KUKA KRL program: MyProgram_097().src

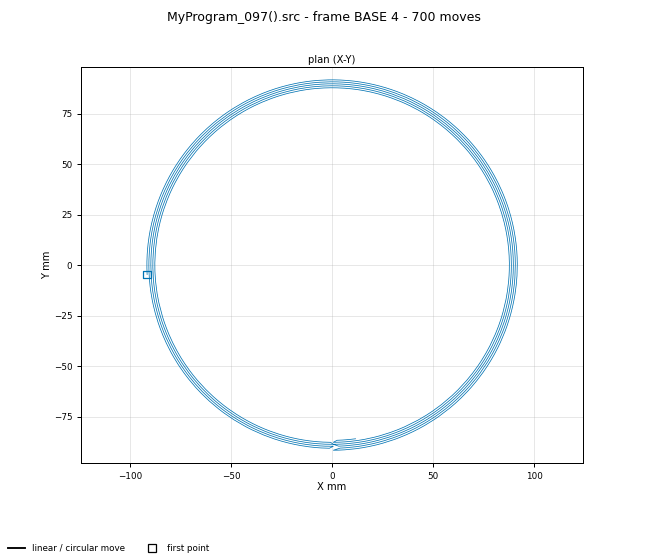
[picture p0: tool path of MyProgram_097().src in frame BASE 4, 700 of 700 moves have a stored position in this frame; points joined in program order, loops and branches not executed]
&ACCESS RVP
&REL 1
&PARAM TEMPLATE = C:\KRC\Roboter\Template\vorgabe
&PARAM EDITMASK = *
DEF MyProgram_097()
; ---- Setting reference (Base) ----
$BASE = BASE_DATA[4]

; --------------------------
; ---- Setting tool (TCP) ----
$TOOL = TOOL_DATA[3]
; --------------------------

$VEL.CP = VEL_APROX_PRINT
Startdeposition()
$VEL.CP = VEL_PRINT
LIN {X -91.5552,Y -4.6883,Z 90,A 177.5634,B 24.9231,C -2.0253,E1 24.8399,E2 -92.3942} C_DIS
LIN {X -91.6643,Y -1.3887,Z 90,A 175.5409,B 24.9225,C -2.0331,E1 24.8398,E2 -90.3782} C_DIS
LIN {X -91.6586,Y 1.702,Z 90,A 173.5845,B 24.9221,C -2.0386,E1 24.8398,E2 -88.423} C_DIS
LIN {X -91.5223,Y 5.2832,Z 90,A 171.2995,B 24.9216,C -2.0444,E1 24.8401,E2 -86.1382} C_DIS
LIN {X -91.3286,Y 7.9677,Z 90,A 169.5918,B 24.9213,C -2.049,E1 24.8405,E2 -84.4312} C_DIS
LIN {X -91.0724,Y 10.4899,Z 90,A 167.9958,B 24.9209,C -2.0538,E1 24.841,E2 -82.837} C_DIS
LIN {X -90.567,Y 14.2076,Z 90,A 165.8073,B 24.92,C -2.0659,E1 24.8419,E2 -80.6644} C_DIS
LIN {X -90.0282,Y 17.295,Z 90,A 163.689,B 24.9198,C -2.0674,E1 24.843,E2 -78.5372} C_DIS
LIN {X -89.2955,Y 20.7489,Z 90,A 161.221,B 24.9199,C -2.0667,E1 24.8445,E2 -76.0529} C_DIS
LIN {X -88.1916,Y 25.0287,Z 90,A 158.7468,B 24.9186,C -2.0839,E1 24.8463,E2 -73.6054} C_DIS
LIN {X -87.1683,Y 28.3884,Z 90,A 155.9671,B 24.9194,C -2.0734,E1 24.8486,E2 -70.7848} C_DIS
LIN {X -86.029,Y 31.6746,Z 90,A 154.4192,B 24.9174,C -2.0987,E1 24.8501,E2 -69.2883} C_DIS
LIN {X -84.932,Y 34.5072,Z 90,A 152.4774,B 24.917,C -2.1032,E1 24.8521,E2 -67.3464} C_DIS
LIN {X -83.7402,Y 37.3084,Z 90,A 150.1569,B 24.9176,C -2.0965,E1 24.8547,E2 -64.9971} C_DIS
LIN {X -81.9719,Y 41.048,Z 90,A 147.8126,B 24.9164,C -2.1113,E1 24.8575,E2 -62.6754} C_DIS
LIN {X -80.4271,Y 43.9975,Z 90,A 145.3042,B 24.9169,C -2.1046,E1 24.8609,E2 -60.138} C_DIS
LIN {X -78.8019,Y 46.8455,Z 90,A 143.8579,B 24.915,C -2.1285,E1 24.8629,E2 -58.7411} C_DIS
LIN {X -77.2171,Y 49.4139,Z 90,A 141.8308,B 24.915,C -2.1296,E1 24.8659,E2 -56.7062} C_DIS
LIN {X -75.2511,Y 52.359,Z 90,A 139.693,B 24.9143,C -2.1379,E1 24.8692,E2 -54.5777} C_DIS
LIN {X -73.255,Y 55.1171,Z 90,A 137.652,B 24.9136,C -2.1463,E1 24.8726,E2 -52.5468} C_DIS
LIN {X -71.7232,Y 57.097,Z 90,A 135.3366,B 24.9151,C -2.1278,E1 24.8767,E2 -50.1765} C_DIS
LIN {X -69.4479,Y 59.8451,Z 90,A 133.6906,B 24.9132,C -2.1511,E1 24.8796,E2 -48.5784} C_DIS
LIN {X -67.0511,Y 62.5179,Z 90,A 131.4415,B 24.9128,C -2.1565,E1 24.8838,E2 -46.3323} C_DIS
LIN {X -64.969,Y 64.6788,Z 90,A 129.4486,B 24.9127,C -2.1575,E1 24.8877,E2 -44.3333} C_DIS
LIN {X -61.8992,Y 67.6216,Z 90,A 126.93,B 24.9118,C -2.168,E1 24.8928,E2 -41.8292} C_DIS
LIN {X -59.0628,Y 70.1145,Z 90,A 124.575,B 24.9114,C -2.1734,E1 24.8978,E2 -39.478} C_DIS
LIN {X -56.7745,Y 71.9782,Z 90,A 122.6887,B 24.9112,C -2.1761,E1 24.9019,E2 -37.5911} C_DIS
LIN {X -53.5559,Y 74.405,Z 90,A 120.329,B 24.9103,C -2.1862,E1 24.9071,E2 -35.2471} C_DIS
LIN {X -51.2942,Y 75.981,Z 90,A 118.4347,B 24.9105,C -2.1844,E1 24.9115,E2 -33.3419} C_DIS
LIN {X -48.8009,Y 77.6063,Z 90,A 116.5005,B 24.9105,C -2.1856,E1 24.9161,E2 -31.4044} C_DIS
LIN {X -44.0262,Y 80.4115,Z 90,A 113.1858,B 24.9095,C -2.1962,E1 24.9241,E2 -28.1052} C_DIS
LIN {X -41.4285,Y 81.78,Z 90,A 111.0703,B 24.91,C -2.1905,E1 24.9293,E2 -25.9703} C_DIS
LIN {X -38.1771,Y 83.3487,Z 90,A 108.4553,B 24.9106,C -2.1828,E1 24.936,E2 -23.3304} C_DIS
LIN {X -34.3452,Y 84.9979,Z 90,A 106.2377,B 24.9093,C -2.1986,E1 24.9417,E2 -21.1455} C_DIS
LIN {X -31.2892,Y 86.1696,Z 90,A 104.1979,B 24.9091,C -2.2015,E1 24.947,E2 -19.1082} C_DIS
LIN {X -28.0201,Y 87.2875,Z 90,A 102.0825,B 24.9088,C -2.2055,E1 24.9526,E2 -16.9983} C_DIS
LIN {X -24.8875,Y 88.2316,Z 90,A 100.0462,B 24.9086,C -2.2079,E1 24.958,E2 -14.9646} C_DIS
LIN {X -21.729,Y 89.062,Z 90,A 97.9504,B 24.9086,C -2.2082,E1 24.9637,E2 -12.8664} C_DIS
LIN {X -18.0864,Y 89.8732,Z 90,A 95.8183,B 24.9078,C -2.2166,E1 24.9695,E2 -10.7517} C_DIS
LIN {X -15.7712,Y 90.3088,Z 90,A 94.2067,B 24.9081,C -2.2133,E1 24.9739,E2 -9.1304} C_DIS
LIN {X -12.884,Y 90.7645,Z 90,A 92.4079,B 24.9079,C -2.2154,E1 24.9789,E2 -7.3352} C_DIS
LIN {X -9.9586,Y 91.1328,Z 90,A 90.491,B 24.908,C -2.214,E1 24.9842,E2 -5.4138} C_DIS
LIN {X -6.8158,Y 91.4219,Z 90,A 87.5202,B 24.9106,C -2.1828,E1 24.9927,E2 -2.3677} C_DIS
LIN {X -1.8331,Y 91.6561,Z 90,A 85.4521,B 24.9078,C -2.2176,E1 24.9982,E2 -0.3819} C_DIS
LIN {X 0.9871,Y 91.67,Z 90,A 83.6399,B 24.9078,C -2.2163,E1 25.0033,E2 1.4333} C_DIS
LIN {X 4.2039,Y 91.5783,Z 90,A 81.6417,B 24.9078,C -2.2169,E1 25.0089,E2 3.4296} C_DIS
LIN {X 7.3964,Y 91.3755,Z 90,A 79.5848,B 24.908,C -2.2149,E1 25.0146,E2 5.4903} C_DIS
LIN {X 10.7821,Y 91.0382,Z 90,A 77.5651,B 24.9077,C -2.2181,E1 25.0202,E2 7.501} C_DIS
LIN {X 14.1056,Y 90.5827,Z 90,A 75.4649,B 24.9077,C -2.2175,E1 25.026,E2 9.6009} C_DIS
LIN {X 17.533,Y 89.9823,Z 90,A 73.3239,B 24.9077,C -2.2177,E1 25.0319,E2 11.7388} C_DIS
LIN {X 20.388,Y 89.3789,Z 90,A 71.448,B 24.908,C -2.2151,E1 25.037,E2 13.6184} C_DIS
LIN {X 23.2363,Y 88.6815,Z 90,A 69.5392,B 24.9083,C -2.2114,E1 25.0422,E2 15.5331} C_DIS
LIN {X 26.6555,Y 87.715,Z 90,A 67.2673,B 24.9085,C -2.2081,E1 25.0483,E2 17.8089} C_DIS
LIN {X 29.2709,Y 86.8758,Z 90,A 65.6725,B 24.9083,C -2.2109,E1 25.0525,E2 19.3942} C_DIS
LIN {X 32.3826,Y 85.7646,Z 90,A 63.643,B 24.9083,C -2.2102,E1 25.0578,E2 21.421} C_DIS
LIN {X 35.1234,Y 84.6806,Z 90,A 61.3887,B 24.9097,C -2.1943,E1 25.0637,E2 23.7079} C_DIS
LIN {X 39.3103,Y 82.8196,Z 90,A 58.6647,B 24.9096,C -2.1957,E1 25.0706,E2 26.4216} C_DIS
LIN {X 42.8304,Y 81.0541,Z 90,A 56.5031,B 24.909,C -2.2028,E1 25.0759,E2 28.5604} C_DIS
LIN {X 45.6049,Y 79.526,Z 90,A 54.4378,B 24.9095,C -2.1971,E1 25.081,E2 30.6331} C_DIS
LIN {X 48.5057,Y 77.7907,Z 90,A 52.3751,B 24.9095,C -2.1957,E1 25.0859,E2 32.6927} C_DIS
LIN {X 51.857,Y 75.5998,Z 90,A 50.0088,B 24.9095,C -2.1963,E1 25.0913,E2 35.0495} C_DIS
LIN {X 55.545,Y 72.9329,Z 90,A 46.9532,B 24.9105,C -2.1841,E1 25.0983,E2 38.1233} C_DIS
LIN {X 58.1956,Y 70.8359,Z 90,A 44.856,B 24.9108,C -2.1807,E1 25.1028,E2 40.2206} C_DIS
LIN {X 60.4754,Y 68.8982,Z 90,A 42.9197,B 24.9113,C -2.1747,E1 25.1069,E2 42.1634} C_DIS
LIN {X 62.7024,Y 66.8777,Z 90,A 41.1502,B 24.9113,C -2.1747,E1 25.1105,E2 43.9256} C_DIS
LIN {X 65.3805,Y 64.2622,Z 90,A 38.9541,B 24.9113,C -2.1749,E1 25.1149,E2 46.1122} C_DIS
LIN {X 67.8006,Y 61.7042,Z 90,A 36.8433,B 24.9114,C -2.1732,E1 25.1189,E2 48.2178} C_DIS
LIN {X 69.4819,Y 59.8052,Z 90,A 35.0348,B 24.9124,C -2.1617,E1 25.1222,E2 50.0454} C_DIS
LIN {X 71.6401,Y 57.202,Z 90,A 32.9262,B 24.9127,C -2.1569,E1 25.126,E2 52.1555} C_DIS
LIN {X 73.8027,Y 54.3823,Z 90,A 30.8163,B 24.9129,C -2.1554,E1 25.1295,E2 54.2588} C_DIS
LIN {X 75.5012,Y 51.9991,Z 90,A 28.8276,B 24.9137,C -2.1451,E1 25.1327,E2 56.262} C_DIS
LIN {X 77.0645,Y 49.6515,Z 90,A 27.2246,B 24.9136,C -2.1463,E1 25.1351,E2 57.8543} C_DIS
LIN {X 78.6827,Y 47.0472,Z 90,A 25.252,B 24.9142,C -2.1392,E1 25.138,E2 59.8335} C_DIS
LIN {X 80.2935,Y 44.2426,Z 90,A 23.2448,B 24.9146,C -2.1343,E1 25.1407,E2 61.8419} C_DIS
LIN {X 82.185,Y 40.618,Z 90,A 20.7535,B 24.9149,C -2.1296,E1 25.1439,E2 64.3311} C_DIS
LIN {X 84.0377,Y 36.6314,Z 90,A 18.297,B 24.9147,C -2.1323,E1 25.1467,E2 66.7679} C_DIS
LIN {X 84.9334,Y 34.5037,Z 90,A 16.6637,B 24.9156,C -2.1213,E1 25.1485,E2 68.4183} C_DIS
LIN {X 86.0757,Y 31.5464,Z 90,A 14.606,B 24.9163,C -2.1127,E1 25.1505,E2 70.4848} C_DIS
LIN {X 87.2488,Y 28.1395,Z 90,A 12.1194,B 24.9175,C -2.0975,E1 25.1527,E2 72.9931} C_DIS
LIN {X 88.4324,Y 24.1654,Z 90,A 9.7762,B 24.9175,C -2.0987,E1 25.1545,E2 75.3202} C_DIS
LIN {X 89.2996,Y 20.7313,Z 90,A 7.6349,B 24.9177,C -2.0945,E1 25.1559,E2 77.4589} C_DIS
LIN {X 90.014,Y 17.3685,Z 90,A 5.5066,B 24.9182,C -2.0886,E1 25.1571,E2 79.5887} C_DIS
LIN {X 90.5925,Y 14.0424,Z 90,A 3.3129,B 24.9189,C -2.079,E1 25.1581,E2 81.7923} C_DIS
LIN {X 91.048,Y 10.6982,Z 90,A 1.3172,B 24.9191,C -2.0765,E1 25.1588,E2 83.7821} C_DIS
LIN {X 91.391,Y 7.2031,Z 90,A -0.8025,B 24.9195,C -2.0722,E1 25.1594,E2 85.8992} C_DIS
LIN {X 91.59,Y 3.9308,Z 90,A -3.3161,B 24.9213,C -2.0488,E1 25.1597,E2 88.4533} C_DIS
LIN {X 91.6732,Y 0.5986,Z 90,A -6.2469,B 24.9241,C -2.0115,E1 25.1597,E2 91.4546} C_DIS
LIN {X 91.5197,Y -5.3293,Z 90,A -9.5373,B 24.9239,C -2.0145,E1 25.1592,E2 94.7184} C_DIS
LIN {X 91.1374,Y -9.9143,Z 90,A -11.3055,B 24.9215,C -2.0455,E1 25.1588,E2 96.4028} C_DIS
LIN {X 90.5357,Y -14.4099,Z 90,A -14.2025,B 24.9224,C -2.0341,E1 25.1577,E2 99.3096} C_DIS
LIN {X 90.0768,Y -17.0424,Z 90,A -16.0185,B 24.9232,C -2.0235,E1 25.1568,E2 101.1402} C_DIS
LIN {X 89.3686,Y -20.4322,Z 90,A -18.1763,B 24.9237,C -2.0168,E1 25.1555,E2 103.301} C_DIS
LIN {X 88.4849,Y -23.9712,Z 90,A -20.3278,B 24.9239,C -2.0143,E1 25.154,E2 105.4461} C_DIS
LIN {X 87.7285,Y -26.6121,Z 90,A -22.2382,B 24.9249,C -2.0018,E1 25.1524,E2 107.3751} C_DIS
LIN {X 86.5823,Y -30.1289,Z 90,A -24.674,B 24.9257,C -1.9902,E1 25.1502,E2 109.8247} C_DIS
LIN {X 85.5227,Y -33.0197,Z 90,A -26.7289,B 24.9265,C -1.9795,E1 25.1482,E2 111.8933} C_DIS
LIN {X 83.3008,Y -38.2801,Z 90,A -29.924,B 24.9263,C -1.9823,E1 25.1446,E2 115.0644} C_DIS
LIN {X 81.986,Y -41.0194,Z 90,A -31.8104,B 24.9267,C -1.9771,E1 25.1423,E2 116.953} C_DIS
LIN {X 80.3066,Y -44.2189,Z 90,A -34.1683,B 24.9275,C -1.9668,E1 25.1392,E2 119.3227} C_DIS
LIN {X 78.5669,Y -47.24,Z 90,A -36.2275,B 24.9276,C -1.9649,E1 25.1363,E2 121.3758} C_DIS
LIN {X 76.7141,Y -50.1921,Z 90,A -38.5472,B 24.9284,C -1.9537,E1 25.1327,E2 123.7105} C_DIS
LIN {X 74.641,Y -53.225,Z 90,A -40.4025,B 24.9277,C -1.9633,E1 25.1298,E2 125.5339} C_DIS
LIN {X 71.7332,Y -57.0844,Z 90,A -43.909,B 24.9296,C -1.9376,E1 25.1238,E2 129.0844} C_DIS
LIN {X 69.0074,Y -60.3505,Z 90,A -46.1494,B 24.929,C -1.9458,E1 25.1198,E2 131.2953} C_DIS
LIN {X 67.0825,Y -62.4845,Z 90,A -48.4727,B 24.9307,C -1.9223,E1 25.1153,E2 133.6638} C_DIS
LIN {X 63.8284,Y -65.8043,Z 90,A -51.6397,B 24.9319,C -1.906,E1 25.109,E2 136.856} C_DIS
LIN {X 60.8838,Y -68.5381,Z 90,A -53.525,B 24.9307,C -1.9225,E1 25.1051,E2 138.6949} C_DIS
LIN {X 58.2099,Y -70.824,Z 90,A -55.808,B 24.9313,C -1.9146,E1 25.1002,E2 140.9878} C_DIS
LIN {X 52.9979,Y -74.8031,Z 90,A -59.5708,B 24.931,C -1.9179,E1 25.0919,E2 144.7293} C_DIS
LIN {X 50.4212,Y -76.563,Z 90,A -61.955,B 24.9324,C -1.8987,E1 25.0862,E2 147.1509} C_DIS
LIN {X 45.896,Y -79.3587,Z 90,A -64.8036,B 24.9317,C -1.9093,E1 25.0795,E2 149.9655} C_DIS
LIN {X 42.9328,Y -81.0001,Z 90,A -67.0077,B 24.9321,C -1.9025,E1 25.0741,E2 152.1792} C_DIS
LIN {X 40.121,Y -82.43,Z 90,A -69.1324,B 24.9328,C -1.8939,E1 25.0687,E2 154.3186} C_DIS
LIN {X 36.7672,Y -83.9785,Z 90,A -72.0004,B 24.9344,C -1.871,E1 25.0613,E2 157.2337} C_DIS
LIN {X 33.1425,Y -85.4747,Z 90,A -73.6168,B 24.9326,C -1.8965,E1 25.0573,E2 158.7862} C_DIS
LIN {X 30.6617,Y -86.3953,Z 90,A -75.7566,B 24.9339,C -1.8775,E1 25.0515,E2 160.9666} C_DIS
LIN {X 25.1022,Y -88.1708,Z 90,A -79.0764,B 24.9334,C -1.8846,E1 25.0427,E2 164.2636} C_DIS
LIN {X 21.9836,Y -88.9999,Z 90,A -81.119,B 24.9336,C -1.8816,E1 25.0372,E2 166.3101} C_DIS
LIN {X 18.4384,Y -89.801,Z 90,A -83.3048,B 24.9336,C -1.8825,E1 25.0312,E2 168.4909} C_DIS
LIN {X 15.0105,Y -90.4372,Z 90,A -85.464,B 24.9336,C -1.8815,E1 25.0253,E2 170.6503} C_DIS
LIN {X 12.0239,Y -90.8827,Z 90,A -88.5954,B 24.9367,C -1.8383,E1 25.0164,E2 173.8814} C_DIS
LIN {X 6.3664,Y -91.4532,Z 90,A -90.8766,B 24.9338,C -1.8793,E1 25.0103,E2 176.0643} C_DIS
LIN {X 3.4384,Y -91.6112,Z 90,A -93.103,B 24.9348,C -1.8653,E1 25.004,E2 178.3232} C_DIS
LIN {X 0.6231,Y -91.6697,Z 90,A -94.7593,B 24.9346,C -1.8684,E1 24.9994,E2 179.972} C_DIS
Enddeposition()
LIN {X 0.6231,Y -91.6697,Z 90,A -94.7593,B 24.9346,C -1.8684,E1 24.9994,E2 179.972} C_DIS
Startdeposition()
$VEL.CP = VEL_PRINT
LIN {X 4.0101,Y -90.6052,Z 90,A -91.6211,B 24.9309,C -1.9197,E1 25.0085,E2 176.7126} C_DIS
LIN {X 6.6191,Y -90.4534,Z 90,A -88.7867,B 24.9279,C -1.9611,E1 25.0167,E2 173.7814} C_DIS
LIN {X 11.8452,Y -89.9172,Z 90,A -86.5115,B 24.9304,C -1.9271,E1 25.0227,E2 171.5887} C_DIS
LIN {X 14.9993,Y -89.4449,Z 90,A -84.194,B 24.9295,C -1.939,E1 25.0292,E2 169.2452} C_DIS
LIN {X 19.6354,Y -88.5433,Z 90,A -81.495,B 24.93,C -1.9318,E1 25.0365,E2 166.5668} C_DIS
LIN {X 22.7552,Y -87.793,Z 90,A -79.7701,B 24.9306,C -1.9234,E1 25.0411,E2 164.8644} C_DIS
LIN {X 25.9972,Y -86.8882,Z 90,A -77.3397,B 24.9297,C -1.9363,E1 25.0477,E2 162.4075} C_DIS
LIN {X 30.4916,Y -85.4149,Z 90,A -74.2799,B 24.9293,C -1.9425,E1 25.0558,E2 159.339} C_DIS
LIN {X 33.6041,Y -84.239,Z 90,A -71.9041,B 24.9283,C -1.9551,E1 25.0621,E2 156.9388} C_DIS
LIN {X 38.4435,Y -82.1432,Z 90,A -68.9672,B 24.929,C -1.9462,E1 25.0695,E2 154.0302} C_DIS
LIN {X 41.5738,Y -80.6046,Z 90,A -67.0434,B 24.9294,C -1.9399,E1 25.0742,E2 152.1263} C_DIS
LIN {X 45.7226,Y -78.3266,Z 90,A -63.8121,B 24.9284,C -1.9537,E1 25.0822,E2 148.872} C_DIS
LIN {X 48.092,Y -76.893,Z 90,A -61.4468,B 24.9266,C -1.979,E1 25.0879,E2 146.4543} C_DIS
LIN {X 51.3642,Y -74.7485,Z 90,A -59.4133,B 24.9274,C -1.9682,E1 25.0925,E2 144.4533} C_DIS
LIN {X 55.8452,Y -71.4628,Z 90,A -56.004,B 24.9271,C -1.972,E1 25.1001,E2 141.0474} C_DIS
LIN {X 59.2143,Y -68.6971,Z 90,A -53.3962,B 24.9271,C -1.9729,E1 25.1056,E2 138.4475} C_DIS
LIN {X 62.5799,Y -65.6442,Z 90,A -50.4365,B 24.9263,C -1.9828,E1 25.1117,E2 135.4763} C_DIS
LIN {X 65.5036,Y -62.7275,Z 90,A -47.7262,B 24.9255,C -1.9929,E1 25.117,E2 132.7539} C_DIS
LIN {X 68.0397,Y -59.9678,Z 90,A -45.7493,B 24.9261,C -1.9847,E1 25.1207,E2 130.8051} C_DIS
LIN {X 71.0974,Y -56.3075,Z 90,A -42.2706,B 24.9243,C -2.0095,E1 25.1269,E2 127.2838} C_DIS
LIN {X 73.2193,Y -53.5192,Z 90,A -40.1284,B 24.924,C -2.0129,E1 25.1305,E2 125.1439} C_DIS
LIN {X 77.1002,Y -47.7604,Z 90,A -36.0628,B 24.924,C -2.0134,E1 25.1367,E2 121.0974} C_DIS
LIN {X 79.5975,Y -43.4705,Z 90,A -32.9008,B 24.9232,C -2.0235,E1 25.1411,E2 117.9281} C_DIS
LIN {X 81.1466,Y -40.5051,Z 90,A -31.0324,B 24.9234,C -2.0207,E1 25.1434,E2 116.0761} C_DIS
LIN {X 82.6228,Y -37.4014,Z 90,A -28.3014,B 24.9214,C -2.0478,E1 25.1467,E2 113.296} C_DIS
LIN {X 84.706,Y -32.4092,Z 90,A -25.4901,B 24.9223,C -2.0359,E1 25.1496,E2 110.5282} C_DIS
LIN {X 85.4964,Y -30.2622,Z 90,A -23.9124,B 24.9216,C -2.0453,E1 25.1511,E2 108.9373} C_DIS
LIN {X 86.468,Y -27.3658,Z 90,A -21.8483,B 24.9207,C -2.0562,E1 25.1529,E2 106.8592} C_DIS
LIN {X 87.4521,Y -24.0345,Z 90,A -19.6811,B 24.9203,C -2.0621,E1 25.1545,E2 104.6905} C_DIS
LIN {X 88.3031,Y -20.6885,Z 90,A -17.5361,B 24.9198,C -2.0677,E1 25.1559,E2 102.5446} C_DIS
LIN {X 88.9645,Y -17.6299,Z 90,A -15.4211,B 24.9189,C -2.079,E1 25.1571,E2 100.4152} C_DIS
LIN {X 89.5913,Y -14.1005,Z 90,A -13.1302,B 24.9183,C -2.0873,E1 25.1582,E2 98.1184} C_DIS
LIN {X 90.1842,Y -9.602,Z 90,A -10.6359,B 24.9187,C -2.0828,E1 25.159,E2 95.6494} C_DIS
LIN {X 90.48,Y -6.2249,Z 90,A -8.41,B 24.9179,C -2.0927,E1 25.1595,E2 93.4131} C_DIS
LIN {X 90.6939,Y 0.4343,Z 90,A -4.3654,B 24.9173,C -2.1001,E1 25.1598,E2 89.3752} C_DIS
LIN {X 90.6247,Y 3.5567,Z 90,A -2.2228,B 24.9163,C -2.1126,E1 25.1596,E2 87.2158} C_DIS
LIN {X 90.425,Y 6.9818,Z 90,A -0.0752,B 24.9158,C -2.1188,E1 25.1592,E2 85.0663} C_DIS
LIN {X 90.0939,Y 10.4156,Z 90,A 2.0687,B 24.9154,C -2.1244,E1 25.1586,E2 82.9219} C_DIS
LIN {X 89.6448,Y 13.755,Z 90,A 4.1631,B 24.9149,C -2.1299,E1 25.1577,E2 80.827} C_DIS
LIN {X 89.0632,Y 17.1206,Z 90,A 6.2893,B 24.9145,C -2.1354,E1 25.1567,E2 78.7001} C_DIS
LIN {X 88.3679,Y 20.4078,Z 90,A 8.4405,B 24.9139,C -2.143,E1 25.1554,E2 76.5435} C_DIS
LIN {X 87.5482,Y 23.6787,Z 90,A 10.6304,B 24.9132,C -2.1517,E1 25.1538,E2 74.3457} C_DIS
LIN {X 85.5548,Y 30.0957,Z 90,A 14.8072,B 24.9123,C -2.1618,E1 25.1503,E2 70.1687} C_DIS
LIN {X 84.3431,Y 33.3414,Z 90,A 18.0714,B 24.9086,C -2.2076,E1 25.1468,E2 66.8145} C_DIS
LIN {X 82.1768,Y 38.3713,Z 90,A 20.4093,B 24.9112,C -2.1763,E1 25.1442,E2 64.5631} C_DIS
LIN {X 81.0584,Y 40.6829,Z 90,A 22.565,B 24.9092,C -2.2001,E1 25.1414,E2 62.3626} C_DIS
LIN {X 79.3997,Y 43.832,Z 90,A 24.3011,B 24.9102,C -2.1876,E1 25.1392,E2 60.6652} C_DIS
LIN {X 77.6517,Y 46.858,Z 90,A 26.4202,B 24.91,C -2.1903,E1 25.1361,E2 58.5506} C_DIS
LIN {X 74.6817,Y 51.4602,Z 90,A 29.8883,B 24.9093,C -2.1994,E1 25.1308,E2 55.0783} C_DIS
LIN {X 72.8822,Y 53.9797,Z 90,A 32.284,B 24.9075,C -2.22,E1 25.1268,E2 52.6455} C_DIS
LIN {X 69.8621,Y 57.8333,Z 90,A 34.8838,B 24.9084,C -2.2097,E1 25.1223,E2 50.0822} C_DIS
LIN {X 67.7151,Y 60.3331,Z 90,A 37.4528,B 24.9066,C -2.2318,E1 25.1175,E2 47.4724} C_DIS
LIN {X 65.478,Y 62.754,Z 90,A 39.0092,B 24.9078,C -2.2176,E1 25.1146,E2 45.9564} C_DIS
LIN {X 63.167,Y 65.08,Z 90,A 41.1612,B 24.9071,C -2.2248,E1 25.1103,E2 43.7964} C_DIS
LIN {X 59.2814,Y 68.6392,Z 90,A 44.4669,B 24.9067,C -2.2306,E1 25.1034,E2 40.4902} C_DIS
LIN {X 56.5778,Y 70.8838,Z 90,A 46.4822,B 24.9069,C -2.2276,E1 25.0991,E2 38.4897} C_DIS
LIN {X 52.8125,Y 73.7309,Z 90,A 49.5888,B 24.9061,C -2.2371,E1 25.0921,E2 35.3717} C_DIS
LIN {X 50.8711,Y 75.0833,Z 90,A 51.8151,B 24.9037,C -2.2652,E1 25.0868,E2 33.0864} C_DIS
LIN {X 47.3894,Y 77.3287,Z 90,A 53.6998,B 24.9056,C -2.2435,E1 25.0825,E2 31.259} C_DIS
LIN {X 44.4638,Y 79.0469,Z 90,A 55.8738,B 24.9052,C -2.2476,E1 25.0772,E2 29.0818} C_DIS
LIN {X 39.5089,Y 81.6363,Z 90,A 59.0311,B 24.9059,C -2.2393,E1 25.0694,E2 25.953} C_DIS
LIN {X 36.6842,Y 82.945,Z 90,A 62.6426,B 24.9009,C -2.2983,E1 25.0599,E2 22.2105} C_DIS
LIN {X 31.0039,Y 85.2299,Z 90,A 65.2073,B 24.9044,C -2.2569,E1 25.0534,E2 19.7492} C_DIS
LIN {X 25.8089,Y 86.9441,Z 90,A 68.6443,B 24.9043,C -2.259,E1 25.0443,E2 16.3138} C_DIS
LIN {X 21.8024,Y 88.0348,Z 90,A 71.2616,B 24.9041,C -2.2604,E1 25.0372,E2 13.6971} C_DIS
LIN {X 18.6353,Y 88.7596,Z 90,A 73.325,B 24.9041,C -2.2618,E1 25.0316,E2 11.6333} C_DIS
LIN {X 15.8129,Y 89.305,Z 90,A 75.1209,B 24.9041,C -2.2618,E1 25.0267,E2 9.8393} C_DIS
LIN {X 12.5979,Y 89.8147,Z 90,A 77.2571,B 24.9038,C -2.265,E1 25.0207,E2 7.6974} C_DIS
LIN {X 9.1211,Y 90.2346,Z 90,A 79.4409,B 24.9038,C -2.2644,E1 25.0147,E2 5.5165} C_DIS
LIN {X 5.6082,Y 90.5217,Z 90,A 81.6746,B 24.9038,C -2.2647,E1 25.0085,E2 3.2832} C_DIS
LIN {X 2.4265,Y 90.6621,Z 90,A 83.6425,B 24.9039,C -2.2631,E1 25.003,E2 1.3196} C_DIS
LIN {X -0.8525,Y 90.6903,Z 90,A 85.5502,B 24.9044,C -2.2573,E1 24.9977,E2 -0.5743} C_DIS
LIN {X -6.1547,Y 90.4848,Z 90,A 89.1019,B 24.904,C -2.2627,E1 24.9878,E2 -4.1396} C_DIS
LIN {X -9.5901,Y 90.1855,Z 90,A 91.2007,B 24.9043,C -2.259,E1 24.9819,E2 -6.2307} C_DIS
LIN {X -12.936,Y 89.7667,Z 90,A 93.3385,B 24.9043,C -2.2579,E1 24.976,E2 -8.3676} C_DIS
LIN {X -16.4969,Y 89.182,Z 90,A 95.8076,B 24.904,C -2.2623,E1 24.9692,E2 -10.8496} C_DIS
LIN {X -21.7149,Y 88.0561,Z 90,A 99.0142,B 24.9047,C -2.2539,E1 24.9605,E2 -14.0404} C_DIS
LIN {X -25.0623,Y 87.1629,Z 90,A 101.2623,B 24.9047,C -2.2535,E1 24.9545,E2 -16.2911} C_DIS
LIN {X -28.2354,Y 86.1873,Z 90,A 103.172,B 24.9054,C -2.2452,E1 24.9494,E2 -18.1843} C_DIS
LIN {X -31.4331,Y 85.0733,Z 90,A 105.7684,B 24.9044,C -2.257,E1 24.9425,E2 -20.814} C_DIS
LIN {X -35.2699,Y 83.5548,Z 90,A 108.5482,B 24.9043,C -2.2588,E1 24.9353,E2 -23.6045} C_DIS
LIN {X -38.2055,Y 82.254,Z 90,A 110.427,B 24.9049,C -2.251,E1 24.9306,E2 -25.4693} C_DIS
LIN {X -42.2329,Y 80.2605,Z 90,A 112.8653,B 24.9064,C -2.2338,E1 24.9246,E2 -27.8732} C_DIS
LIN {X -44.9691,Y 78.7605,Z 90,A 115.5563,B 24.9048,C -2.2529,E1 24.9179,E2 -30.6177} C_DIS
LIN {X -48.1319,Y 76.8681,Z 90,A 117.352,B 24.9066,C -2.2319,E1 24.9138,E2 -32.3689} C_DIS
LIN {X -51.111,Y 74.9208,Z 90,A 119.63,B 24.9068,C -2.2284,E1 24.9085,E2 -34.6463} C_DIS
LIN {X -57.0594,Y 70.4954,Z 90,A 124.9245,B 24.9061,C -2.2375,E1 24.8967,E2 -39.9817} C_DIS
LIN {X -60.1037,Y 67.9204,Z 90,A 126.7859,B 24.9083,C -2.2115,E1 24.8929,E2 -41.7883} C_DIS
LIN {X -64.3952,Y 63.8644,Z 90,A 130.4846,B 24.9091,C -2.2017,E1 24.8855,E2 -45.4791} C_DIS
LIN {X -67.7274,Y 60.3194,Z 90,A 133.5631,B 24.9097,C -2.1942,E1 24.8796,E2 -48.5531} C_DIS
LIN {X -71.8006,Y 55.408,Z 90,A 137.5857,B 24.9106,C -2.1834,E1 24.8726,E2 -52.5688} C_DIS
LIN {X -74.177,Y 52.1861,Z 90,A 140.2703,B 24.9108,C -2.1812,E1 24.8681,E2 -55.2611} C_DIS
LIN {X -75.9626,Y 49.5506,Z 90,A 142.2804,B 24.9112,C -2.1756,E1 24.865,E2 -57.2679} C_DIS
LIN {X -78.1296,Y 46.056,Z 90,A 145.7127,B 24.9097,C -2.1936,E1 24.8601,E2 -60.7608} C_DIS
LIN {X -80.3289,Y 42.1032,Z 90,A 147.6875,B 24.9126,C -2.1585,E1 24.8576,E2 -62.6623} C_DIS
LIN {X -82.7728,Y 37.0686,Z 90,A 151.3379,B 24.9132,C -2.1514,E1 24.8532,E2 -66.3155} C_DIS
LIN {X -84.0685,Y 34.0277,Z 90,A 153.4026,B 24.9138,C -2.1443,E1 24.851,E2 -68.375} C_DIS
LIN {X -85.3828,Y 30.5819,Z 90,A 155.9969,B 24.9137,C -2.1451,E1 24.8485,E2 -70.9858} C_DIS
LIN {X -87.4382,Y 24.0859,Z 90,A 159.8645,B 24.9158,C -2.1186,E1 24.8454,E2 -74.8123} C_DIS
LIN {X -88.4416,Y 20.0888,Z 90,A 162.8121,B 24.9157,C -2.1206,E1 24.8434,E2 -77.782} C_DIS
LIN {X -89.1791,Y 16.5128,Z 90,A 165.0907,B 24.9163,C -2.1124,E1 24.8422,E2 -80.0545} C_DIS
LIN {X -89.7357,Y 13.154,Z 90,A 167.1485,B 24.9171,C -2.1028,E1 24.8413,E2 -82.1015} C_DIS
LIN {X -90.052,Y 10.7728,Z 90,A 169.0581,B 24.9165,C -2.1097,E1 24.8406,E2 -84.0391} C_DIS
LIN {X -90.3994,Y 7.3025,Z 90,A 171.3029,B 24.917,C -2.1038,E1 24.8401,E2 -86.2835} C_DIS
LIN {X -90.6517,Y 2.7643,Z 90,A 173.7513,B 24.9187,C -2.082,E1 24.8398,E2 -88.6943} C_DIS
LIN {X -90.6961,Y -0.1334,Z 90,A 175.5206,B 24.9193,C -2.0742,E1 24.8398,E2 -90.4558} C_DIS
LIN {X -90.6456,Y -2.9638,Z 90,A 177.6408,B 24.919,C -2.0785,E1 24.8399,E2 -92.5989} C_DIS
LIN {X -90.4326,Y -6.8874,Z 90,A -179.9745,B 24.9198,C -2.0676,E1 24.8404,E2 -94.9722} C_DIS
LIN {X -90.0869,Y -10.4747,Z 90,A -178.1518,B 24.9214,C -2.0469,E1 24.8409,E2 -96.7563} C_DIS
LIN {X -89.7585,Y -12.9938,Z 90,A -175.8787,B 24.9203,C -2.0618,E1 24.8418,E2 -99.0787} C_DIS
LIN {X -89.0257,Y -17.3153,Z 90,A -173.3012,B 24.9214,C -2.0475,E1 24.8431,E2 -101.6371} C_DIS
LIN {X -88.4092,Y -20.229,Z 90,A -170.8113,B 24.9204,C -2.0601,E1 24.8446,E2 -104.1718} C_DIS
LIN {X -87.5006,Y -23.855,Z 90,A -169.068,B 24.9224,C -2.0342,E1 24.8458,E2 -105.8633} C_DIS
LIN {X -86.1294,Y -28.4141,Z 90,A -165.9451,B 24.9228,C -2.0286,E1 24.8484,E2 -108.9909} C_DIS
LIN {X -84.9731,Y -31.7039,Z 90,A -163.7615,B 24.9234,C -2.0216,E1 24.8505,E2 -111.1701} C_DIS
LIN {X -83.6662,Y -35.0056,Z 90,A -161.5335,B 24.9239,C -2.0147,E1 24.8529,E2 -113.394} C_DIS
LIN {X -82.1057,Y -38.524,Z 90,A -159.384,B 24.9251,C -1.9993,E1 24.8553,E2 -115.5185} C_DIS
LIN {X -79.9421,Y -42.8345,Z 90,A -156.0014,B 24.9249,C -2.001,E1 24.8596,E2 -118.9235} C_DIS
LIN {X -78.4967,Y -45.4281,Z 90,A -153.958,B 24.9249,C -2.0012,E1 24.8625,E2 -120.9778} C_DIS
LIN {X -76.3508,Y -48.9483,Z 90,A -151.5621,B 24.9259,C -1.988,E1 24.866,E2 -123.3546} C_DIS
LIN {X -75.1669,Y -50.7477,Z 90,A -149.6153,B 24.9248,C -2.0027,E1 24.8691,E2 -125.346} C_DIS
LIN {X -73.1597,Y -53.6007,Z 90,A -147.3135,B 24.925,C -2.0003,E1 24.8729,E2 -127.6534} C_DIS
LIN {X -70.8116,Y -56.6692,Z 90,A -145.6493,B 24.9272,C -1.9704,E1 24.8757,E2 -129.254} C_DIS
LIN {X -67.4517,Y -60.6274,Z 90,A -142.1672,B 24.9273,C -1.9691,E1 24.8821,E2 -132.7489} C_DIS
LIN {X -65.0354,Y -63.2132,Z 90,A -140.173,B 24.9282,C -1.9568,E1 24.8859,E2 -134.7223} C_DIS
LIN {X -60.7805,Y -67.3145,Z 90,A -136.1808,B 24.9282,C -1.9572,E1 24.894,E2 -138.732} C_DIS
LIN {X -56.0648,Y -71.2893,Z 90,A -132.2571,B 24.9287,C -1.9507,E1 24.9024,E2 -142.6553} C_DIS
LIN {X -53.5433,Y -73.2017,Z 90,A -128.9797,B 24.9259,C -1.9883,E1 24.9101,E2 -146.0337} C_DIS
LIN {X -48.5013,Y -76.6373,Z 90,A -126.3377,B 24.9292,C -1.9431,E1 24.916,E2 -148.5767} C_DIS
LIN {X -42.7863,Y -79.9686,Z 90,A -122.3691,B 24.9301,C -1.9305,E1 24.9256,E2 -152.5271} C_DIS
LIN {X -39.7033,Y -81.5429,Z 90,A -118.5786,B 24.9265,C -1.9803,E1 24.9355,E2 -156.4456} C_DIS
LIN {X -33.6949,Y -84.204,Z 90,A -115.8428,B 24.9302,C -1.9294,E1 24.9422,E2 -159.0667} C_DIS
LIN {X -28.6323,Y -86.0563,Z 90,A -112.4262,B 24.9304,C -1.9269,E1 24.9512,E2 -162.484} C_DIS
LIN {X -25.083,Y -87.1571,Z 90,A -110.0708,B 24.9304,C -1.9255,E1 24.9575,E2 -164.84} C_DIS
LIN {X -21.7148,Y -88.0562,Z 90,A -107.9032,B 24.9307,C -1.9231,E1 24.9633,E2 -167.005} C_DIS
LIN {X -18.5617,Y -88.7747,Z 90,A -105.8691,B 24.9307,C -1.9218,E1 24.9689,E2 -169.0387} C_DIS
LIN {X -15.327,Y -89.3901,Z 90,A -103.6726,B 24.9305,C -1.925,E1 24.975,E2 -171.245} C_DIS
LIN {X -11.3177,Y -89.9855,Z 90,A -101.1457,B 24.9306,C -1.9233,E1 24.9819,E2 -173.7699} C_DIS
LIN {X -7.9972,Y -90.3412,Z 90,A -99.0942,B 24.9308,C -1.9212,E1 24.9876,E2 -175.8175} C_DIS
LIN {X -5.4523,Y -90.5309,Z 90,A -97.1199,B 24.9299,C -1.9335,E1 24.9932,E2 -177.8215} C_DIS
LIN {X -1.3463,Y -90.6844,Z 90,A -93.7922,B 24.9281,C -1.9589,E1 25.0027,E2 -181.2098} C_DIS
LIN {X -1.3463,Y -90.6844,Z 90,A -93.7922,B 24.9281,C -1.9589,E1 25.0027,E2 -181.2098} C_DIS
Enddeposition()
LIN {X 0.5962,Y -89.6879,Z 90,A -93.8733,B 24.93,C -1.932,E1 25.0023,E2 -181.0649} C_DIS
Startdeposition()
$VEL.CP = VEL_PRINT
LIN {X -3.4183,Y -89.6492,Z 90,A -97.0165,B 24.9315,C -1.912,E1 24.9934,E2 -177.8739} C_DIS
LIN {X -6.2141,Y -89.498,Z 90,A -98.895,B 24.9317,C -1.9089,E1 24.9881,E2 -175.9877} C_DIS
LIN {X -9.2198,Y -89.2384,Z 90,A -100.9097,B 24.9319,C -1.9062,E1 24.9825,E2 -173.9654} C_DIS
LIN {X -12.7845,Y -88.7979,Z 90,A -103.2694,B 24.932,C -1.9045,E1 24.9759,E2 -171.5999} C_DIS
LIN {X -16.1805,Y -88.2426,Z 90,A -105.4894,B 24.932,C -1.9045,E1 24.9698,E2 -169.3777} C_DIS
LIN {X -19.6314,Y -87.5406,Z 90,A -107.7281,B 24.932,C -1.9058,E1 24.9637,E2 -167.1394} C_DIS
LIN {X -22.8707,Y -86.7508,Z 90,A -109.8874,B 24.9319,C -1.9061,E1 24.9579,E2 -164.9776} C_DIS
LIN {X -26.836,Y -85.606,Z 90,A -112.2545,B 24.9311,C -1.9165,E1 24.9516,E2 -162.6312} C_DIS
LIN {X -30.9069,Y -84.2216,Z 90,A -115.2492,B 24.9315,C -1.9109,E1 24.9436,E2 -159.6175} C_DIS
LIN {X -35.577,Y -82.358,Z 90,A -118.9673,B 24.9324,C -1.8983,E1 24.934,E2 -155.8611} C_DIS
LIN {X -38.7182,Y -80.9284,Z 90,A -120.5264,B 24.9308,C -1.921,E1 24.9301,E2 -154.3519} C_DIS
LIN {X -41.6056,Y -79.4827,Z 90,A -122.3907,B 24.9302,C -1.9297,E1 24.9255,E2 -152.5034} C_DIS
LIN {X -46.1138,Y -76.956,Z 90,A -125.84,B 24.9302,C -1.9296,E1 24.9172,E2 -149.0436} C_DIS
LIN {X -49.6468,Y -74.7246,Z 90,A -129.3131,B 24.9317,C -1.909,E1 24.9089,E2 -145.5104} C_DIS
LIN {X -52.7173,Y -72.5913,Z 90,A -131.0119,B 24.9299,C -1.9341,E1 24.9051,E2 -143.8654} C_DIS
LIN {X -55.1167,Y -70.7872,Z 90,A -133.5041,B 24.9309,C -1.92,E1 24.8995,E2 -141.3304} C_DIS
LIN {X -57.6536,Y -68.736,Z 90,A -135.2038,B 24.9298,C -1.9355,E1 24.8959,E2 -139.6612} C_DIS
LIN {X -60.5397,Y -66.2076,Z 90,A -137.8457,B 24.9298,C -1.9346,E1 24.8904,E2 -137.0065} C_DIS
LIN {X -64.3229,Y -62.5395,Z 90,A -140.6902,B 24.9282,C -1.9573,E1 24.8849,E2 -134.2043} C_DIS
LIN {X -68.0417,Y -58.4718,Z 90,A -144.719,B 24.9287,C -1.9499,E1 24.8773,E2 -130.1397} C_DIS
LIN {X -70.5831,Y -55.377,Z 90,A -147.5366,B 24.9288,C -1.9482,E1 24.8723,E2 -127.3049} C_DIS
LIN {X -72.5386,Y -52.7892,Z 90,A -149.6888,B 24.9286,C -1.9509,E1 24.8688,E2 -125.1487} C_DIS
LIN {X -74.5633,Y -49.8902,Z 90,A -151.4741,B 24.9272,C -1.9706,E1 24.8661,E2 -123.4014} C_DIS
LIN {X -76.4288,Y -46.9822,Z 90,A -153.7428,B 24.9269,C -1.9745,E1 24.8627,E2 -121.1304} C_DIS
LIN {X -77.7978,Y -44.6764,Z 90,A -155.3399,B 24.9263,C -1.9824,E1 24.8605,E2 -119.5441} C_DIS
LIN {X -79.7572,Y -41.0768,Z 90,A -158.3418,B 24.9266,C -1.9783,E1 24.8565,E2 -116.5163} C_DIS
LIN {X -82.2439,Y -35.8388,Z 90,A -161.7371,B 24.9252,C -1.9977,E1 24.8526,E2 -113.1488} C_DIS
LIN {X -83.5677,Y -32.6336,Z 90,A -163.9542,B 24.9247,C -2.004,E1 24.8503,E2 -110.9344} C_DIS
LIN {X -84.8331,Y -29.1912,Z 90,A -166.3828,B 24.9244,C -2.0084,E1 24.848,E2 -108.5024} C_DIS
LIN {X -86.4287,Y -24.057,Z 90,A -169.6534,B 24.9232,C -2.0234,E1 24.8454,E2 -105.2489} C_DIS
LIN {X -87.5941,Y -19.3861,Z 90,A -172.7876,B 24.9226,C -2.0311,E1 24.8433,E2 -102.1147} C_DIS
LIN {X -88.1951,Y -16.4429,Z 90,A -175.3443,B 24.9236,C -2.0186,E1 24.842,E2 -99.513} C_DIS
LIN {X -88.7667,Y -13.0039,Z 90,A -177.3967,B 24.9227,C -2.0306,E1 24.8411,E2 -97.477} C_DIS
LIN {X -89.2141,Y -9.4521,Z 90,A -179.3027,B 24.9213,C -2.0488,E1 24.8405,E2 -95.6029} C_DIS
LIN {X -89.511,Y -6.021,Z 90,A 178.0484,B 24.9217,C -2.0428,E1 24.84,E2 -92.9238} C_DIS
LIN {X -89.7153,Y 0.1667,Z 90,A 174.407,B 24.9201,C -2.0644,E1 24.8398,E2 -89.3121} C_DIS
LIN {X -89.6479,Y 3.4479,Z 90,A 171.6269,B 24.9211,C -2.0515,E1 24.8401,E2 -86.4845} C_DIS
LIN {X -89.3963,Y 7.5457,Z 90,A 170.0116,B 24.9182,C -2.0888,E1 24.8404,E2 -84.9485} C_DIS
LIN {X -88.9214,Y 11.8996,Z 90,A 166.8965,B 24.9182,C -2.0886,E1 24.8414,E2 -81.8142} C_DIS
LIN {X -88.4376,Y 15.078,Z 90,A 164.7783,B 24.9178,C -2.0932,E1 24.8423,E2 -79.6945} C_DIS
LIN {X -87.5853,Y 19.4268,Z 90,A 162.1186,B 24.9167,C -2.1071,E1 24.8438,E2 -77.0523} C_DIS
LIN {X -86.8782,Y 22.3755,Z 90,A 160.0775,B 24.9165,C -2.1102,E1 24.8452,E2 -75.0067} C_DIS
LIN {X -85.9527,Y 25.7033,Z 90,A 157.5858,B 24.9165,C -2.1089,E1 24.8471,E2 -72.4974} C_DIS
LIN {X -84.7316,Y 29.4805,Z 90,A 154.8813,B 24.9164,C -2.1119,E1 24.8496,E2 -69.7846} C_DIS
LIN {X -83.4418,Y 32.9542,Z 90,A 152.8171,B 24.9151,C -2.1278,E1 24.8516,E2 -67.7468} C_DIS
LIN {X -81.8054,Y 36.8287,Z 90,A 149.9711,B 24.9148,C -2.1313,E1 24.8548,E2 -64.8934} C_DIS
LIN {X -80.4624,Y 39.6776,Z 90,A 148.1938,B 24.9138,C -2.144,E1 24.857,E2 -63.1369} C_DIS
LIN {X -77.899,Y 44.5003,Z 90,A 144.9154,B 24.9125,C -2.1603,E1 24.8613,E2 -59.8799} C_DIS
LIN {X -75.5078,Y 48.4464,Z 90,A 141.8747,B 24.912,C -2.1659,E1 24.8657,E2 -56.837} C_DIS
LIN {X -74.121,Y 50.5434,Z 90,A 139.9221,B 24.9125,C -2.1601,E1 24.8688,E2 -54.861} C_DIS
LIN {X -71.4106,Y 54.3073,Z 90,A 137.0127,B 24.9117,C -2.1696,E1 24.8736,E2 -51.9602} C_DIS
LIN {X -68.0229,Y 58.4938,Z 90,A 133.7766,B 24.9105,C -2.1846,E1 24.8793,E2 -48.7447} C_DIS
LIN {X -64.8668,Y 61.9742,Z 90,A 130.6236,B 24.9102,C -2.1875,E1 24.8853,E2 -45.5849} C_DIS
LIN {X -60.4989,Y 66.2451,Z 90,A 126.8956,B 24.9091,C -2.2019,E1 24.8927,E2 -41.8755} C_DIS
LIN {X -57.2995,Y 69.0307,Z 90,A 124.0905,B 24.9088,C -2.2051,E1 24.8987,E2 -39.0671} C_DIS
LIN {X -55.1009,Y 70.7993,Z 90,A 121.5099,B 24.9104,C -2.1858,E1 24.9045,E2 -36.431} C_DIS
LIN {X -52.1116,Y 73.0264,Z 90,A 119.9629,B 24.9079,C -2.2154,E1 24.9078,E2 -34.9493} C_DIS
LIN {X -49.9654,Y 74.5124,Z 90,A 117.6651,B 24.9092,C -2.1998,E1 24.9132,E2 -32.6066} C_DIS
LIN {X -45.6209,Y 77.2477,Z 90,A 114.5411,B 24.9083,C -2.2105,E1 24.9206,E2 -29.4983} C_DIS
LIN {X -42.9807,Y 78.7477,Z 90,A 112.7481,B 24.9077,C -2.2182,E1 24.925,E2 -27.7185} C_DIS
LIN {X -38.7414,Y 80.9172,Z 90,A 109.4515,B 24.9079,C -2.2153,E1 24.9333,E2 -24.4064} C_DIS
LIN {X -35.1472,Y 82.5425,Z 90,A 107.2495,B 24.9068,C -2.2286,E1 24.9388,E2 -22.2309} C_DIS
LIN {X -30.1641,Y 84.4917,Z 90,A 103.2407,B 24.908,C -2.2151,E1 24.9494,E2 -18.1815} C_DIS
LIN {X -26.7733,Y 85.6254,Z 90,A 101.7132,B 24.9058,C -2.2409,E1 24.9533,E2 -16.7128} C_DIS
LIN {X -24.2028,Y 86.3873,Z 90,A 99.3566,B 24.9073,C -2.2228,E1 24.9598,E2 -14.3094} C_DIS
LIN {X -21.0985,Y 87.1973,Z 90,A 97.6522,B 24.9063,C -2.2354,E1 24.9643,E2 -12.6326} C_DIS
LIN {X -16.2951,Y 88.222,Z 90,A 94.6088,B 24.9058,C -2.2409,E1 24.9726,E2 -9.5987} C_DIS
LIN {X -13.0651,Y 88.758,Z 90,A 92.501,B 24.9058,C -2.2418,E1 24.9785,E2 -7.4912} C_DIS
LIN {X -9.6011,Y 89.1985,Z 90,A 90.3455,B 24.9054,C -2.2455,E1 24.9844,E2 -5.3428} C_DIS
LIN {X -5.4922,Y 89.5457,Z 90,A 87.1944,B 24.9067,C -2.2303,E1 24.9933,E2 -2.1545} C_DIS
LIN {X -2.2073,Y 89.6878,Z 90,A 85.5309,B 24.9055,C -2.2446,E1 24.9978,E2 -0.5249} C_DIS
LIN {X 0.9272,Y 89.7093,Z 90,A 83.4427,B 24.9057,C -2.2423,E1 25.0037,E2 1.5688} C_DIS
LIN {X 4.2434,Y 89.6138,Z 90,A 81.4195,B 24.9054,C -2.2455,E1 25.0093,E2 3.5838} C_DIS
LIN {X 7.6129,Y 89.3909,Z 90,A 79.2184,B 24.9055,C -2.244,E1 25.0154,E2 5.7875} C_DIS
LIN {X 11.0972,Y 89.0254,Z 90,A 77.0086,B 24.9055,C -2.2445,E1 25.0216,E2 7.9945} C_DIS
LIN {X 14.0797,Y 88.6024,Z 90,A 74.991,B 24.9058,C -2.2409,E1 25.0272,E2 10.0187} C_DIS
LIN {X 17.446,Y 88.002,Z 90,A 72.83,B 24.9058,C -2.2407,E1 25.0331,E2 12.1776} C_DIS
LIN {X 20.8896,Y 87.2482,Z 90,A 70.314,B 24.9066,C -2.2309,E1 25.04,E2 14.7133} C_DIS
LIN {X 24.9613,Y 86.1723,Z 90,A 67.5442,B 24.907,C -2.2265,E1 25.0474,E2 17.489} C_DIS
LIN {X 29.5914,Y 84.6926,Z 90,A 64.5304,B 24.907,C -2.2269,E1 25.0554,E2 20.496} C_DIS
LIN {X 35.7271,Y 82.2926,Z 90,A 60.732,B 24.9062,C -2.2361,E1 25.0651,E2 24.2639} C_DIS
LIN {X 39.1724,Y 80.7102,Z 90,A 57.1402,B 24.9097,C -2.1945,E1 25.0744,E2 27.9449} C_DIS
LIN {X 44.0927,Y 78.1312,Z 90,A 54.1253,B 24.9086,C -2.2072,E1 25.0816,E2 30.9208} C_DIS
LIN {X 47.3238,Y 76.2168,Z 90,A 51.971,B 24.9082,C -2.2117,E1 25.0867,E2 33.0575} C_DIS
LIN {X 50.6103,Y 74.0758,Z 90,A 49.8181,B 24.9076,C -2.2195,E1 25.0917,E2 35.1848} C_DIS
LIN {X 56.1697,Y 69.9544,Z 90,A 45.7119,B 24.9074,C -2.2224,E1 25.1008,E2 39.2694} C_DIS
LIN {X 61.5906,Y 65.2312,Z 90,A 41.284,B 24.9076,C -2.219,E1 25.1101,E2 43.6877} C_DIS
LIN {X 63.1282,Y 63.7442,Z 90,A 39.5813,B 24.9088,C -2.2046,E1 25.1135,E2 45.4175} C_DIS
LIN {X 67.6288,Y 58.9478,Z 90,A 35.7054,B 24.9087,C -2.2065,E1 25.1208,E2 49.2718} C_DIS
LIN {X 69.127,Y 57.1837,Z 90,A 33.0212,B 24.9124,C -2.1614,E1 25.1258,E2 52.0502} C_DIS
LIN {X 71.9597,Y 53.5764,Z 90,A 30.9634,B 24.9105,C -2.1843,E1 25.1291,E2 54.044} C_DIS
LIN {X 73.8522,Y 50.9357,Z 90,A 28.4841,B 24.9121,C -2.1651,E1 25.1331,E2 56.5567} C_DIS
LIN {X 77.0754,Y 45.9125,Z 90,A 25.4189,B 24.9108,C -2.1813,E1 25.1376,E2 59.5682} C_DIS
LIN {X 80.0919,Y 40.4224,Z 90,A 21.1326,B 24.9125,C -2.1603,E1 25.1434,E2 63.8816} C_DIS
LIN {X 81.4745,Y 37.5565,Z 90,A 18.2408,B 24.9154,C -2.1245,E1 25.1468,E2 66.8422} C_DIS
LIN {X 83.2847,Y 33.3479,Z 90,A 16.1185,B 24.9138,C -2.1442,E1 25.149,E2 68.9064} C_DIS
LIN {X 84.4571,Y 30.2613,Z 90,A 13.1499,B 24.9167,C -2.1078,E1 25.1519,E2 71.9442} C_DIS
LIN {X 85.9724,Y 25.6368,Z 90,A 11.4361,B 24.9135,C -2.1476,E1 25.1532,E2 73.5542} C_DIS
LIN {X 87.2669,Y 20.813,Z 90,A 7.7987,B 24.9156,C -2.122,E1 25.1558,E2 77.2312} C_DIS
LIN {X 87.9909,Y 17.5039,Z 90,A 5.6081,B 24.9162,C -2.1143,E1 25.157,E2 79.4272} C_DIS
LIN {X 88.6244,Y 13.9371,Z 90,A 3.4057,B 24.9164,C -2.1111,E1 25.1581,E2 81.6243} C_DIS
LIN {X 89.0945,Y 10.519,Z 90,A 1.2348,B 24.9169,C -2.1053,E1 25.1588,E2 83.796} C_DIS
LIN {X 89.4348,Y 7.0646,Z 90,A -1.0079,B 24.9175,C -2.0973,E1 25.1594,E2 86.0442} C_DIS
LIN {X 89.6406,Y 3.6183,Z 90,A -3.2135,B 24.9181,C -2.0903,E1 25.1597,E2 88.2534} C_DIS
LIN {X 89.7156,Y 0.1318,Z 90,A -6.111,B 24.9205,C -2.0593,E1 25.1597,E2 91.2066} C_DIS
LIN {X 89.6291,Y -3.8867,Z 90,A -7.9518,B 24.9191,C -2.0769,E1 25.1596,E2 92.995} C_DIS
LIN {X 89.4097,Y -7.3787,Z 90,A -10.2371,B 24.9198,C -2.0679,E1 25.1591,E2 95.288} C_DIS
LIN {X 88.9397,Y -11.7588,Z 90,A -12.8043,B 24.9198,C -2.0677,E1 25.1583,E2 97.8406} C_DIS
LIN {X 88.647,Y -13.7912,Z 90,A -14.1409,B 24.9202,C -2.0626,E1 25.1577,E2 99.1813} C_DIS
LIN {X 87.8434,Y -18.2222,Z 90,A -17.2376,B 24.9215,C -2.0455,E1 25.1561,E2 102.3001} C_DIS
LIN {X 87.2268,Y -20.9773,Z 90,A -18.8943,B 24.9215,C -2.045,E1 25.155,E2 103.9484} C_DIS
LIN {X 86.35,Y -24.3346,Z 90,A -21.0698,B 24.922,C -2.0395,E1 25.1535,E2 106.1244} C_DIS
LIN {X 85.2537,Y -27.9357,Z 90,A -23.7624,B 24.9234,C -2.0217,E1 25.1512,E2 108.8438} C_DIS
LIN {X 83.7057,Y -32.282,Z 90,A -27.2835,B 24.9256,C -1.9923,E1 25.1476,E2 112.4147} C_DIS
LIN {X 81.9461,Y -36.5166,Z 90,A -29.9347,B 24.9256,C -1.9932,E1 25.1446,E2 115.0492} C_DIS
LIN {X 80.3675,Y -39.8692,Z 90,A -31.4282,B 24.9237,C -2.0172,E1 25.1429,E2 116.4782} C_DIS
LIN {X 79.1756,Y -42.1887,Z 90,A -33.9212,B 24.9263,C -1.9829,E1 25.1396,E2 119.0389} C_DIS
LIN {X 77.3936,Y -45.3741,Z 90,A -35.5826,B 24.925,C -1.9999,E1 25.1373,E2 120.6517} C_DIS
LIN {X 75.5824,Y -48.3302,Z 90,A -38.2413,B 24.9267,C -1.9779,E1 25.1333,E2 123.3489} C_DIS
LIN {X 71.7787,Y -53.8173,Z 90,A -42.2311,B 24.9268,C -1.9759,E1 25.1268,E2 127.324} C_DIS
LIN {X 68.9625,Y -57.3816,Z 90,A -45.1967,B 24.9275,C -1.966,E1 25.1216,E2 130.2993} C_DIS
LIN {X 65.5468,Y -61.255,Z 90,A -48.6789,B 24.9286,C -1.9512,E1 25.115,E2 133.8009} C_DIS
LIN {X 61.0445,Y -65.7431,Z 90,A -52.3855,B 24.9284,C -1.9538,E1 25.1076,E2 137.4858} C_DIS
LIN {X 57.3542,Y -68.9853,Z 90,A -55.7137,B 24.9294,C -1.9401,E1 25.1005,E2 140.8335} C_DIS
LIN {X 53.5571,Y -71.9742,Z 90,A -59.0227,B 24.9305,C -1.9259,E1 25.0931,E2 144.1641} C_DIS
LIN {X 50.6997,Y -74.0152,Z 90,A -61.3852,B 24.9311,C -1.9173,E1 25.0877,E2 146.5389} C_DIS
LIN {X 47.4578,Y -76.133,Z 90,A -63.0492,B 24.9294,C -1.9404,E1 25.0839,E2 148.1429} C_DIS
LIN {X 45.6312,Y -77.2416,Z 90,A -65.4516,B 24.9322,C -1.9024,E1 25.0779,E2 150.6279} C_DIS
LIN {X 41.4424,Y -79.5686,Z 90,A -67.4238,B 24.9299,C -1.9342,E1 25.0732,E2 152.5191} C_DIS
LIN {X 38.8977,Y -80.8422,Z 90,A -69.7945,B 24.9314,C -1.9124,E1 25.0672,E2 154.9352} C_DIS
LIN {X 35.4598,Y -82.4083,Z 90,A -71.9805,B 24.9311,C -1.9165,E1 25.0616,E2 157.1062} C_DIS
LIN {X 31.813,Y -83.8833,Z 90,A -74.9322,B 24.9325,C -1.8982,E1 25.0538,E2 160.0948} C_DIS
LIN {X 28.2163,Y -85.1614,Z 90,A -76.6591,B 24.931,C -1.9191,E1 25.0494,E2 161.7688} C_DIS
LIN {X 22.9098,Y -86.7403,Z 90,A -80.3346,B 24.9316,C -1.9105,E1 25.0395,E2 165.4586} C_DIS
LIN {X 19.6707,Y -87.5317,Z 90,A -82.5055,B 24.9318,C -1.907,E1 25.0336,E2 167.6346} C_DIS
LIN {X 15.5938,Y -88.3482,Z 90,A -84.6622,B 24.9308,C -1.9216,E1 25.0278,E2 169.7543} C_DIS
LIN {X 12.1418,Y -88.8892,Z 90,A -87.4876,B 24.9323,C -1.9002,E1 25.0198,E2 172.6278} C_DIS
LIN {X 6.5013,Y -89.4786,Z 90,A -90.88,B 24.9319,C -1.9059,E1 25.0105,E2 176.0046} C_DIS
LIN {X 3.2748,Y -89.655,Z 90,A -93.7471,B 24.9338,C -1.8788,E1 25.0023,E2 178.9351} C_DIS
LIN {X 3.2748,Y -89.655,Z 90,A -93.7471,B 24.9338,C -1.8788,E1 25.0023,E2 178.9351} C_DIS
Enddeposition()
LIN {X 0.5879,Y -88.7176,Z 90,A -94.1059,B 24.9294,C -1.9401,E1 25.0017,E2 179.1485} C_DIS
Startdeposition()
$VEL.CP = VEL_PRINT
LIN {X 3.8467,Y -88.6494,Z 90,A -91.6962,B 24.9287,C -1.9506,E1 25.0085,E2 176.7144} C_DIS
LIN {X 6.8081,Y -88.4716,Z 90,A -89.9549,B 24.929,C -1.9457,E1 25.0133,E2 174.9856} C_DIS
LIN {X 11.7253,Y -87.9553,Z 90,A -86.4624,B 24.9282,C -1.9575,E1 25.0231,E2 171.4675} C_DIS
LIN {X 15.119,Y -87.4366,Z 90,A -84.4733,B 24.9286,C -1.9515,E1 25.0285,E2 169.4946} C_DIS
LIN {X 17.2901,Y -87.0316,Z 90,A -82.4188,B 24.9269,C -1.974,E1 25.0343,E2 167.3894} C_DIS
LIN {X 20.4747,Y -86.3398,Z 90,A -80.7153,B 24.9278,C -1.9623,E1 25.0388,E2 165.7158} C_DIS
LIN {X 22.8105,Y -85.7514,Z 90,A -78.7868,B 24.9267,C -1.9767,E1 25.0441,E2 163.7564} C_DIS
LIN {X 27.1367,Y -84.4816,Z 90,A -76.5799,B 24.9283,C -1.9561,E1 25.0499,E2 161.6023} C_DIS
LIN {X 31.5872,Y -82.9204,Z 90,A -73.3736,B 24.9276,C -1.9655,E1 25.0583,E2 158.3803} C_DIS
LIN {X 33.887,Y -82.0085,Z 90,A -71.4963,B 24.9267,C -1.9773,E1 25.0632,E2 156.4793} C_DIS
LIN {X 37.4546,Y -80.4404,Z 90,A -68.9623,B 24.9264,C -1.9818,E1 25.0697,E2 153.941} C_DIS
LIN {X 40.6955,Y -78.8512,Z 90,A -66.5505,B 24.9259,C -1.9885,E1 25.0757,E2 151.52} C_DIS
LIN {X 45.2049,Y -76.3546,Z 90,A -63.5363,B 24.9262,C -1.9835,E1 25.083,E2 148.5266} C_DIS
LIN {X 49.873,Y -73.3909,Z 90,A -60.3718,B 24.9268,C -1.9763,E1 25.0904,E2 145.3894} C_DIS
LIN {X 51.9364,Y -71.9465,Z 90,A -58.1447,B 24.925,C -2.0005,E1 25.0955,E2 143.1128} C_DIS
LIN {X 54.5168,Y -70.0116,Z 90,A -56.4157,B 24.9256,C -1.9925,E1 25.0993,E2 141.4089} C_DIS
LIN {X 58.7828,Y -66.4709,Z 90,A -52.8097,B 24.9249,C -2.0014,E1 25.107,E2 137.7959} C_DIS
LIN {X 61.322,Y -64.1336,Z 90,A -50.4769,B 24.9242,C -2.0104,E1 25.1118,E2 135.4514} C_DIS
LIN {X 63.9158,Y -61.549,Z 90,A -47.5657,B 24.9223,C -2.0356,E1 25.1175,E2 132.4932} C_DIS
LIN {X 66.4264,Y -58.8325,Z 90,A -45.9534,B 24.9239,C -2.014,E1 25.1205,E2 130.939} C_DIS
LIN {X 69.2691,Y -55.4562,Z 90,A -42.9193,B 24.9229,C -2.028,E1 25.1259,E2 127.8858} C_DIS
LIN {X 71.7294,Y -52.2347,Z 90,A -40.1295,B 24.9219,C -2.0412,E1 25.1306,E2 125.0782} C_DIS
LIN {X 73.3633,Y -49.9137,Z 90,A -37.9672,B 24.9206,C -2.0581,E1 25.134,E2 122.8867} C_DIS
LIN {X 75.281,Y -46.971,Z 90,A -36.6198,B 24.9226,C -2.0316,E1 25.1359,E2 121.6087} C_DIS
LIN {X 77.7824,Y -42.7028,Z 90,A -32.9193,B 24.9205,C -2.0589,E1 25.1411,E2 117.863} C_DIS
LIN {X 79.1502,Y -40.1103,Z 90,A -31.1725,B 24.9205,C -2.0592,E1 25.1433,E2 116.1246} C_DIS
LIN {X 81.3803,Y -35.3662,Z 90,A -27.2922,B 24.9183,C -2.0872,E1 25.1479,E2 112.1993} C_DIS
LIN {X 82.7402,Y -32.0583,Z 90,A -25.4616,B 24.9191,C -2.077,E1 25.1497,E2 110.4029} C_DIS
LIN {X 83.7576,Y -29.2948,Z 90,A -23.5685,B 24.9187,C -2.0826,E1 25.1515,E2 108.5073} C_DIS
LIN {X 84.962,Y -25.5931,Z 90,A -21.1761,B 24.9184,C -2.0861,E1 25.1535,E2 106.1202} C_DIS
LIN {X 85.9056,Y -22.2206,Z 90,A -19.3361,B 24.919,C -2.0781,E1 25.1548,E2 104.3096} C_DIS
LIN {X 86.7143,Y -18.8186,Z 90,A -16.7032,B 24.9174,C -2.0987,E1 25.1565,E2 101.6433} C_DIS
LIN {X 87.3398,Y -15.6609,Z 90,A -14.579,B 24.9167,C -2.107,E1 25.1576,E2 99.512} C_DIS
LIN {X 88.2051,Y -9.6726,Z 90,A -10.6813,B 24.9158,C -2.1191,E1 25.159,E2 95.6087} C_DIS
LIN {X 88.5251,Y -6.0679,Z 90,A -8.4095,B 24.9154,C -2.1243,E1 25.1595,E2 93.3382} C_DIS
LIN {X 88.6776,Y -3.1607,Z 90,A -6.0951,B 24.9136,C -2.146,E1 25.1598,E2 90.9863} C_DIS
LIN {X 88.7353,Y 0.1058,Z 90,A -4.2402,B 24.9138,C -2.1435,E1 25.1598,E2 89.1483} C_DIS
LIN {X 88.6357,Y 4.1649,Z 90,A -1.7927,B 24.9137,C -2.1456,E1 25.1595,E2 86.7103} C_DIS
LIN {X 88.4097,Y 7.5821,Z 90,A 0.425,B 24.9131,C -2.1529,E1 25.159,E2 84.4887} C_DIS
LIN {X 88.0292,Y 11.1549,Z 90,A 2.6205,B 24.9128,C -2.1558,E1 25.1583,E2 82.2994} C_DIS
LIN {X 87.5777,Y 14.2752,Z 90,A 4.7102,B 24.9122,C -2.1641,E1 25.1574,E2 80.2024} C_DIS
LIN {X 86.9319,Y 17.7865,Z 90,A 6.9122,B 24.9119,C -2.1675,E1 25.1563,E2 78.0051} C_DIS
LIN {X 86.1753,Y 21.1503,Z 90,A 8.9867,B 24.9118,C -2.1689,E1 25.155,E2 75.9393} C_DIS
LIN {X 85.637,Y 23.2341,Z 90,A 10.7207,B 24.9104,C -2.1855,E1 25.1537,E2 74.1762} C_DIS
LIN {X 84.2146,Y 27.9541,Z 90,A 13.8913,B 24.9097,C -2.1945,E1 25.151,E2 71.0023} C_DIS
LIN {X 82.8921,Y 31.6618,Z 90,A 15.9481,B 24.9105,C -2.1847,E1 25.1491,E2 68.98} C_DIS
LIN {X 80.7116,Y 36.8693,Z 90,A 19.923,B 24.9087,C -2.2068,E1 25.1447,E2 64.9749} C_DIS
LIN {X 79.1241,Y 40.1615,Z 90,A 23.0663,B 24.9058,C -2.2412,E1 25.1407,E2 61.767} C_DIS
LIN {X 76.9744,Y 44.1414,Z 90,A 25.0736,B 24.9078,C -2.2166,E1 25.138,E2 59.8283} C_DIS
LIN {X 75.7965,Y 46.1346,Z 90,A 27.5372,B 24.9046,C -2.2548,E1 25.1343,E2 57.2868} C_DIS
LIN {X 73.1576,Y 50.217,Z 90,A 29.7791,B 24.9066,C -2.231,E1 25.1309,E2 55.1123} C_DIS
LIN {X 71.1413,Y 53.0333,Z 90,A 33.1623,B 24.9027,C -2.277,E1 25.1251,E2 51.6366} C_DIS
LIN {X 67.575,Y 57.5076,Z 90,A 35.3195,B 24.9066,C -2.2316,E1 25.1214,E2 49.5967} C_DIS
LIN {X 62.9365,Y 62.5506,Z 90,A 40.0309,B 24.9049,C -2.2512,E1 25.1124,E2 44.8596} C_DIS
LIN {X 59.1962,Y 66.1008,Z 90,A 43.7157,B 24.9033,C -2.2702,E1 25.1048,E2 41.1448} C_DIS
LIN {X 56.1047,Y 68.7449,Z 90,A 47.0572,B 24.9008,C -2.2999,E1 25.0975,E2 37.7458} C_DIS
LIN {X 51.8574,Y 72.0033,Z 90,A 49.3988,B 24.9036,C -2.2674,E1 25.0924,E2 35.4894} C_DIS
LIN {X 49.3718,Y 73.7302,Z 90,A 51.1316,B 24.9039,C -2.263,E1 25.0884,E2 33.7727} C_DIS
LIN {X 44.4592,Y 76.7917,Z 90,A 55.076,B 24.9028,C -2.2756,E1 25.079,E2 29.8109} C_DIS
LIN {X 42.4996,Y 77.8931,Z 90,A 57.2478,B 24.9006,C -2.302,E1 25.0735,E2 27.5829} C_DIS
LIN {X 38.8359,Y 79.784,Z 90,A 59.2632,B 24.9022,C -2.2834,E1 25.0686,E2 25.6171} C_DIS
LIN {X 35.6917,Y 81.2384,Z 90,A 61.1994,B 24.9028,C -2.2759,E1 25.0637,E2 23.7034} C_DIS
LIN {X 30.3565,Y 83.3786,Z 90,A 65.159,B 24.9018,C -2.2877,E1 25.0534,E2 19.7245} C_DIS
LIN {X 27.5592,Y 84.3449,Z 90,A 67.1654,B 24.9014,C -2.2925,E1 25.048,E2 17.7108} C_DIS
LIN {X 23.549,Y 85.5519,Z 90,A 70.2568,B 24.9001,C -2.3071,E1 25.0396,E2 14.5897} C_DIS
LIN {X 20.2385,Y 86.3944,Z 90,A 71.9357,B 24.9015,C -2.291,E1 25.0352,E2 12.9516} C_DIS
LIN {X 16.4075,Y 87.2035,Z 90,A 74.5773,B 24.9011,C -2.2958,E1 25.0279,E2 10.3018} C_DIS
LIN {X 12.6763,Y 87.8229,Z 90,A 76.8639,B 24.9015,C -2.2914,E1 25.0217,E2 8.0277} C_DIS
LIN {X 9.3882,Y 88.2349,Z 90,A 78.994,B 24.9015,C -2.2914,E1 25.0158,E2 5.899} C_DIS
LIN {X 6.0677,Y 88.5251,Z 90,A 81.1146,B 24.9015,C -2.2906,E1 25.0099,E2 3.7815} C_DIS
LIN {X 2.7811,Y 88.6892,Z 90,A 83.2228,B 24.9016,C -2.2899,E1 25.004,E2 1.6756} C_DIS
LIN {X -0.4706,Y 88.7316,Z 90,A 85.4238,B 24.9014,C -2.2928,E1 24.9978,E2 -0.5321} C_DIS
LIN {X -4.8261,Y 88.6015,Z 90,A 88.6765,B 24.9002,C -2.3059,E1 24.9887,E2 -3.8167} C_DIS
LIN {X -9.7507,Y 88.1969,Z 90,A 91.2761,B 24.902,C -2.2855,E1 24.9816,E2 -6.3691} C_DIS
LIN {X -12.6481,Y 87.8269,Z 90,A 93.337,B 24.9016,C -2.2898,E1 24.9758,E2 -8.442} C_DIS
LIN {X -16.2946,Y 87.2252,Z 90,A 96.2355,B 24.9004,C -2.3042,E1 24.9678,E2 -11.3776} C_DIS
LIN {X -19.6352,Y 86.5337,Z 90,A 97.7736,B 24.9024,C -2.2813,E1 24.9637,E2 -12.8633} C_DIS
LIN {X -24.1427,Y 85.3853,Z 90,A 100.8859,B 24.9024,C -2.2817,E1 24.9553,E2 -15.9812} C_DIS
LIN {X -26.2131,Y 84.7726,Z 90,A 102.7915,B 24.9011,C -2.2961,E1 24.9501,E2 -17.9242} C_DIS
LIN {X -29.2988,Y 83.7562,Z 90,A 104.8775,B 24.9013,C -2.2931,E1 24.9446,E2 -20.0072} C_DIS
LIN {X -34.1012,Y 81.9193,Z 90,A 107.5633,B 24.9034,C -2.269,E1 24.9378,E2 -22.6413} C_DIS
LIN {X -40.6403,Y 78.8794,Z 90,A 112.4555,B 24.9034,C -2.2689,E1 24.9254,E2 -27.5458} C_DIS
LIN {X -43.715,Y 77.2189,Z 90,A 114.4891,B 24.9043,C -2.2582,E1 24.9205,E2 -29.5598} C_DIS
LIN {X -46.2413,Y 75.7317,Z 90,A 116.2681,B 24.9049,C -2.2514,E1 24.9162,E2 -31.328} C_DIS
LIN {X -50.2162,Y 73.1581,Z 90,A 119.6408,B 24.9046,C -2.2549,E1 24.9083,E2 -34.7203} C_DIS
LIN {X -53.0689,Y 71.1142,Z 90,A 122.4249,B 24.9037,C -2.266,E1 24.902,E2 -37.5404} C_DIS
LIN {X -55.6749,Y 69.0932,Z 90,A 124.3192,B 24.9047,C -2.2543,E1 24.8979,E2 -39.4139} C_DIS
LIN {X -59.5224,Y 65.8088,Z 90,A 127.0803,B 24.9066,C -2.2318,E1 24.8922,E2 -42.1324} C_DIS
LIN {X -62.1363,Y 63.3458,Z 90,A 129.8185,B 24.906,C -2.2388,E1 24.8866,E2 -44.8986} C_DIS
LIN {X -65.169,Y 60.2213,Z 90,A 132.8669,B 24.906,C -2.239,E1 24.8807,E2 -47.9606} C_DIS
LIN {X -67.3104,Y 57.8182,Z 90,A 134.878,B 24.9066,C -2.2316,E1 24.8771,E2 -49.9634} C_DIS
LIN {X -69.8512,Y 54.7216,Z 90,A 137.1157,B 24.908,C -2.2145,E1 24.8732,E2 -52.1708} C_DIS
LIN {X -71.929,Y 51.9596,Z 90,A 139.6666,B 24.9077,C -2.2179,E1 24.869,E2 -54.7421} C_DIS
LIN {X -74.1599,Y 48.7221,Z 90,A 142.0188,B 24.9088,C -2.2054,E1 24.8653,E2 -57.0762} C_DIS
LIN {X -76.5029,Y 44.954,Z 90,A 144.6886,B 24.9099,C -2.1916,E1 24.8615,E2 -59.7266} C_DIS
LIN {X -78.7906,Y 40.8141,Z 90,A 148.0202,B 24.9099,C -2.1908,E1 24.857,E2 -63.074} C_DIS
LIN {X -80.3303,Y 37.6913,Z 90,A 150.107,B 24.9109,C -2.1794,E1 24.8545,E2 -65.1449} C_DIS
LIN {X -82.0013,Y 33.9048,Z 90,A 152.9682,B 24.9111,C -2.1768,E1 24.8514,E2 -68.0158} C_DIS
LIN {X -84.0752,Y 28.3704,Z 90,A 156.6389,B 24.9124,C -2.1608,E1 24.8479,E2 -71.6691} C_DIS
LIN {X -85.1955,Y 24.8081,Z 90,A 159.2575,B 24.9125,C -2.1593,E1 24.8457,E2 -74.2992} C_DIS
LIN {X -86.1108,Y 21.4149,Z 90,A 161.8136,B 24.9125,C -2.1606,E1 24.8439,E2 -76.8731} C_DIS
LIN {X -86.9882,Y 17.5101,Z 90,A 164.2681,B 24.9134,C -2.1486,E1 24.8425,E2 -79.3134} C_DIS
LIN {X -87.7698,Y 13.0473,Z 90,A 168.0667,B 24.9121,C -2.1649,E1 24.8409,E2 -83.1736} C_DIS
LIN {X -88.3696,Y 8.0216,Z 90,A 169.7342,B 24.9167,C -2.1077,E1 24.8405,E2 -84.7145} C_DIS
LIN {X -88.6996,Y 2.4424,Z 90,A 173.7976,B 24.9166,C -2.1091,E1 24.8398,E2 -88.8059} C_DIS
LIN {X -88.727,Y -1.0627,Z 90,A 176.3238,B 24.9166,C -2.1095,E1 24.8398,E2 -91.3482} C_DIS
LIN {X -88.4636,Y -6.908,Z 90,A -179.9907,B 24.9177,C -2.0948,E1 24.8404,E2 -95.0207} C_DIS
LIN {X -88.2525,Y -9.22,Z 90,A -177.8226,B 24.9165,C -2.1097,E1 24.8411,E2 -97.2373} C_DIS
LIN {X -87.7749,Y -13.0139,Z 90,A -175.8306,B 24.9182,C -2.0879,E1 24.8418,E2 -99.1891} C_DIS
LIN {X -86.9744,Y -17.5796,Z 90,A -173.1796,B 24.9198,C -2.0686,E1 24.8432,E2 -101.8099} C_DIS
LIN {X -86.473,Y -19.8983,Z 90,A -170.7271,B 24.918,C -2.091,E1 24.8447,E2 -104.3302} C_DIS
LIN {X -85.4962,Y -23.7512,Z 90,A -168.4159,B 24.9192,C -2.0756,E1 24.8464,E2 -106.6181} C_DIS
LIN {X -84.0904,Y -28.3252,Z 90,A -165.8634,B 24.9211,C -2.0506,E1 24.8486,E2 -109.1255} C_DIS
LIN {X -83.0977,Y -31.1191,Z 90,A -163.7977,B 24.9212,C -2.0494,E1 24.8505,E2 -111.2001} C_DIS
LIN {X -81.8192,Y -34.3386,Z 90,A -161.833,B 24.9223,C -2.035,E1 24.8526,E2 -113.1413} C_DIS
LIN {X -80.6737,Y -36.9531,Z 90,A -159.6031,B 24.9219,C -2.0411,E1 24.8552,E2 -115.3982} C_DIS
LIN {X -79.5676,Y -39.275,Z 90,A -157.5863,B 24.9214,C -2.0472,E1 24.8577,E2 -117.4402} C_DIS
LIN {X -77.395,Y -43.3998,Z 90,A -155.0429,B 24.9231,C -2.0251,E1 24.861,E2 -119.9444} C_DIS
LIN {X -76.1125,Y -45.6145,Z 90,A -153.1781,B 24.923,C -2.027,E1 24.8637,E2 -121.8234} C_DIS
LIN {X -74.1615,Y -48.7197,Z 90,A -151.1803,B 24.9243,C -2.0099,E1 24.8667,E2 -123.7904} C_DIS
LIN {X -70.8385,Y -53.4363,Z 90,A -147.1202,B 24.9242,C -2.0107,E1 24.8733,E2 -127.8722} C_DIS
LIN {X -68.5813,Y -56.3062,Z 90,A -145.0052,B 24.9252,C -1.9978,E1 24.877,E2 -129.9664} C_DIS
LIN {X -64.6872,Y -60.7378,Z 90,A -141.2452,B 24.9259,C -1.9877,E1 24.8839,E2 -133.7192} C_DIS
LIN {X -61.4101,Y -64.0497,Z 90,A -137.5031,B 24.9247,C -2.0038,E1 24.8915,E2 -137.5154} C_DIS
LIN {X -59.0567,Y -66.2257,Z 90,A -135.8451,B 24.926,C -1.987,E1 24.8948,E2 -139.1401} C_DIS
LIN {X -56.9894,Y -68.0136,Z 90,A -133.4757,B 24.9248,C -2.0024,E1 24.9,E2 -141.5551} C_DIS
LIN {X -54.0484,Y -70.3725,Z 90,A -131.6464,B 24.9265,C -1.9793,E1 24.9039,E2 -143.3361} C_DIS
LIN {X -51.89,Y -71.98,Z 90,A -128.9658,B 24.9246,C -2.0057,E1 24.9102,E2 -146.089} C_DIS
LIN {X -47.8954,Y -74.6963,Z 90,A -126.7742,B 24.9271,C -1.9718,E1 24.9151,E2 -148.207} C_DIS
LIN {X -45.1279,Y -76.4002,Z 90,A -124.9978,B 24.9281,C -1.9587,E1 24.9193,E2 -149.9577} C_DIS
LIN {X -41.7067,Y -78.3213,Z 90,A -122.0999,B 24.9275,C -1.9666,E1 24.9265,E2 -152.8828} C_DIS
LIN {X -38.657,Y -79.8699,Z 90,A -120.1394,B 24.9283,C -1.9562,E1 24.9313,E2 -154.8236} C_DIS
LIN {X -33.3402,Y -82.2311,Z 90,A -116.1065,B 24.9279,C -1.9608,E1 24.9417,E2 -158.8771} C_DIS
LIN {X -30.4907,Y -83.3297,Z 90,A -114.1137,B 24.9279,C -1.9597,E1 24.9469,E2 -160.8714} C_DIS
LIN {X -26.6157,Y -84.6477,Z 90,A -111.5069,B 24.9282,C -1.9565,E1 24.9538,E2 -163.4753} C_DIS
LIN {X -23.2513,Y -85.6323,Z 90,A -109.2672,B 24.9284,C -1.9543,E1 24.9598,E2 -165.7132} C_DIS
LIN {X -20.0542,Y -86.4369,Z 90,A -107.1975,B 24.9286,C -1.9512,E1 24.9655,E2 -167.7786} C_DIS
LIN {X -16.8625,Y -87.1158,Z 90,A -105.0471,B 24.9286,C -1.9518,E1 24.9713,E2 -169.9327} C_DIS
LIN {X -13.3106,Y -87.7291,Z 90,A -102.8813,B 24.929,C -1.9459,E1 24.9773,E2 -172.0865} C_DIS
LIN {X -10.4465,Y -88.1158,Z 90,A -100.8714,B 24.9287,C -1.9502,E1 24.9829,E2 -174.1081} C_DIS
LIN {X -7.3845,Y -88.4255,Z 90,A -98.8238,B 24.9286,C -1.952,E1 24.9886,E2 -176.1611} C_DIS
LIN {X -3.4203,Y -88.6677,Z 90,A -95.9994,B 24.9279,C -1.9608,E1 24.9965,E2 -179.007} C_DIS
LIN {X 0.5879,Y -88.7176,Z 90,A -94.1027,B 24.9295,C -1.9388,E1 25.0017,E2 -180.8515} C_DIS
Enddeposition()
LIN {X 0.5879,Y -88.7176,Z 90,A -94.1027,B 24.9295,C -1.9388,E1 25.0017,E2 -180.8515} C_DIS
Startdeposition()
$VEL.CP = VEL_PRINT
LIN {X -0.7273,Y -87.7495,Z 90,A -95.7393,B 24.9301,C -1.9304,E1 24.9971,E2 -179.195} C_DIS
LIN {X -4.4986,Y -87.6376,Z 90,A -98.101,B 24.9299,C -1.9334,E1 24.9905,E2 -176.8399} C_DIS
LIN {X -7.8115,Y -87.4043,Z 90,A -100.2346,B 24.9299,C -1.9345,E1 24.9846,E2 -174.7082} C_DIS
LIN {X -10.9204,Y -87.0709,Z 90,A -102.3393,B 24.9299,C -1.9328,E1 24.9787,E2 -172.598} C_DIS
LIN {X -14.202,Y -86.5958,Z 90,A -104.3927,B 24.9297,C -1.9369,E1 24.9731,E2 -170.5525} C_DIS
LIN {X -17.1454,Y -86.0625,Z 90,A -106.3893,B 24.9297,C -1.9363,E1 24.9676,E2 -168.5521} C_DIS
LIN {X -20.2837,Y -85.3775,Z 90,A -108.5193,B 24.9297,C -1.9363,E1 24.9618,E2 -166.4194} C_DIS
LIN {X -22.7525,Y -84.7514,Z 90,A -110.8037,B 24.931,C -1.9181,E1 24.9555,E2 -164.0884} C_DIS
LIN {X -26.4288,Y -83.6791,Z 90,A -113.1044,B 24.9305,C -1.926,E1 24.9494,E2 -161.8025} C_DIS
LIN {X -31.0313,Y -82.0824,Z 90,A -115.7144,B 24.929,C -1.9464,E1 24.9426,E2 -159.2356} C_DIS
LIN {X -33.798,Y -80.983,Z 90,A -118.2881,B 24.9302,C -1.9291,E1 24.9359,E2 -156.615} C_DIS
LIN {X -36.7838,Y -79.6711,Z 90,A -119.9364,B 24.929,C -1.9461,E1 24.9318,E2 -155.0031} C_DIS
LIN {X -38.9206,Y -78.6489,Z 90,A -121.5071,B 24.929,C -1.9472,E1 24.9278,E2 -153.4309} C_DIS
LIN {X -41.4488,Y -77.3476,Z 90,A -123.3444,B 24.9287,C -1.9502,E1 24.9233,E2 -151.5956} C_DIS
LIN {X -44.3925,Y -75.6958,Z 90,A -125.5849,B 24.9286,C -1.9521,E1 24.9179,E2 -149.3531} C_DIS
LIN {X -47.4058,Y -73.8455,Z 90,A -127.7217,B 24.9279,C -1.9608,E1 24.9128,E2 -147.2303} C_DIS
LIN {X -51.0607,Y -71.3672,Z 90,A -130.7889,B 24.9279,C -1.96,E1 24.9058,E2 -144.1508} C_DIS
LIN {X -53.1798,Y -69.8041,Z 90,A -132.7546,B 24.9283,C -1.9556,E1 24.9014,E2 -142.1675} C_DIS
LIN {X -56.3439,Y -67.2751,Z 90,A -135.1792,B 24.9275,C -1.9671,E1 24.8961,E2 -139.7611} C_DIS
LIN {X -58.9274,Y -65.0254,Z 90,A -138.4355,B 24.9293,C -1.9416,E1 24.8893,E2 -136.4311} C_DIS
LIN {X -62.5436,Y -61.5531,Z 90,A -140.7255,B 24.9267,C -1.9771,E1 24.8849,E2 -134.216} C_DIS
LIN {X -66.6981,Y -57.025,Z 90,A -144.7356,B 24.926,C -1.9862,E1 24.8774,E2 -130.2095} C_DIS
LIN {X -68.8422,Y -54.4171,Z 90,A -146.7937,B 24.9253,C -1.9956,E1 24.8738,E2 -128.1643} C_DIS
LIN {X -70.6722,Y -52.0187,Z 90,A -148.542,B 24.9245,C -2.0068,E1 24.8709,E2 -126.4344} C_DIS
LIN {X -72.9888,Y -48.7169,Z 90,A -151.5903,B 24.9249,C -2.0013,E1 24.866,E2 -123.358} C_DIS
LIN {X -74.7912,Y -45.9008,Z 90,A -153.8338,B 24.9246,C -2.0053,E1 24.8627,E2 -121.1125} C_DIS
LIN {X -76.8202,Y -42.418,Z 90,A -156.338,B 24.9238,C -2.0159,E1 24.8592,E2 -118.6206} C_DIS
LIN {X -78.8696,Y -38.4749,Z 90,A -159.2625,B 24.9232,C -2.0232,E1 24.8555,E2 -115.698} C_DIS
LIN {X -80.8364,Y -34.146,Z 90,A -162.4332,B 24.9227,C -2.0302,E1 24.8519,E2 -112.5263} C_DIS
LIN {X -81.9618,Y -31.3497,Z 90,A -164.3974,B 24.9223,C -2.036,E1 24.8499,E2 -110.565} C_DIS
LIN {X -82.9797,Y -28.5502,Z 90,A -166.3931,B 24.9219,C -2.0402,E1 24.8481,E2 -108.5681} C_DIS
LIN {X -83.8997,Y -25.7173,Z 90,A -168.5464,B 24.9219,C -2.0402,E1 24.8463,E2 -106.4022} C_DIS
LIN {X -85.7523,Y -18.6281,Z 90,A -172.9651,B 24.92,C -2.0651,E1 24.8433,E2 -102.0173} C_DIS
LIN {X -86.6196,Y -14.06,Z 90,A -176.0405,B 24.9194,C -2.0734,E1 24.8417,E2 -98.9434} C_DIS
LIN {X -87.3777,Y -8.0996,Z 90,A -179.6855,B 24.9178,C -2.0936,E1 24.8405,E2 -95.3248} C_DIS
LIN {X -87.6998,Y -3.057,Z 90,A 176.5697,B 24.918,C -2.0914,E1 24.8399,E2 -91.5522} C_DIS
LIN {X -87.7474,Y 1.0712,Z 90,A 173.8509,B 24.9173,C -2.0993,E1 24.8399,E2 -88.8361} C_DIS
LIN {X -87.4597,Y 7.1623,Z 90,A 170.0072,B 24.916,C -2.116,E1 24.8404,E2 -85.009} C_DIS
LIN {X -86.753,Y 13.2068,Z 90,A 165.9776,B 24.9151,C -2.127,E1 24.8418,E2 -80.9817} C_DIS
LIN {X -85.8719,Y 18.0739,Z 90,A 162.3658,B 24.9151,C -2.1266,E1 24.8437,E2 -77.3473} C_DIS
LIN {X -85.0925,Y 21.4452,Z 90,A 160.169,B 24.9145,C -2.1354,E1 24.8451,E2 -75.1589} C_DIS
LIN {X -84.2405,Y 24.5796,Z 90,A 158.2123,B 24.9136,C -2.1467,E1 24.8466,E2 -73.2177} C_DIS
LIN {X -83.2814,Y 27.6556,Z 90,A 156.17,B 24.9129,C -2.1549,E1 24.8483,E2 -71.1834} C_DIS
LIN {X -81.6528,Y 32.1447,Z 90,A 152.9964,B 24.9123,C -2.1629,E1 24.8514,E2 -68.011} C_DIS
LIN {X -80.201,Y 35.6159,Z 90,A 150.3065,B 24.9122,C -2.1638,E1 24.8543,E2 -65.3081} C_DIS
LIN {X -78.8958,Y 38.4204,Z 90,A 148.2377,B 24.9118,C -2.1684,E1 24.8568,E2 -63.239} C_DIS
LIN {X -77.7189,Y 40.7463,Z 90,A 146.3901,B 24.9118,C -2.1693,E1 24.8592,E2 -61.3838} C_DIS
LIN {X -75.4657,Y 44.7819,Z 90,A 143.0837,B 24.9117,C -2.1698,E1 24.8639,E2 -58.0615} C_DIS
LIN {X -73.697,Y 47.6371,Z 90,A 141.5143,B 24.9097,C -2.1936,E1 24.8662,E2 -56.5408} C_DIS
LIN {X -71.6455,Y 50.6696,Z 90,A 138.6385,B 24.9103,C -2.1863,E1 24.8708,E2 -53.6336} C_DIS
LIN {X -67.4455,Y 56.1389,Z 90,A 134.4603,B 24.9086,C -2.2074,E1 24.8779,E2 -49.4861} C_DIS
LIN {X -65.4796,Y 58.4201,Z 90,A 131.8552,B 24.9097,C -2.1942,E1 24.8829,E2 -46.8377} C_DIS
LIN {X -62.9404,Y 61.1481,Z 90,A 130.0107,B 24.9078,C -2.2169,E1 24.8863,E2 -45.0394} C_DIS
LIN {X -60.454,Y 63.6064,Z 90,A 127.5533,B 24.9078,C -2.2173,E1 24.8913,E2 -42.5727} C_DIS
LIN {X -57.8205,Y 66.0096,Z 90,A 125.3007,B 24.9072,C -2.2248,E1 24.896,E2 -40.329} C_DIS
LIN {X -54.9869,Y 68.3887,Z 90,A 122.7661,B 24.907,C -2.2266,E1 24.9014,E2 -37.7891} C_DIS
LIN {X -50.6674,Y 71.6479,Z 90,A 119.5526,B 24.9056,C -2.2432,E1 24.9086,E2 -34.6037} C_DIS
LIN {X -46.9796,Y 74.1188,Z 90,A 116.3871,B 24.9058,C -2.2409,E1 24.916,E2 -31.4224} C_DIS
LIN {X -43.9577,Y 75.949,Z 90,A 114.1707,B 24.9052,C -2.2477,E1 24.9213,E2 -29.2155} C_DIS
LIN {X -41.0881,Y 77.5389,Z 90,A 112.0681,B 24.9048,C -2.2525,E1 24.9265,E2 -27.1184} C_DIS
LIN {X -38.7596,Y 78.7287,Z 90,A 109.5486,B 24.9066,C -2.2313,E1 24.9329,E2 -24.542} C_DIS
LIN {X -34.9394,Y 80.4967,Z 90,A 107.5268,B 24.9045,C -2.2568,E1 24.938,E2 -22.5758} C_DIS
LIN {X -30.0175,Y 82.4585,Z 90,A 104.0383,B 24.9041,C -2.2605,E1 24.947,E2 -19.0888} C_DIS
LIN {X -26.7855,Y 83.5647,Z 90,A 101.8412,B 24.9038,C -2.2642,E1 24.9528,E2 -16.8963} C_DIS
LIN {X -23.4581,Y 84.5601,Z 90,A 99.7805,B 24.9031,C -2.2729,E1 24.9583,E2 -14.8528} C_DIS
LIN {X -21.3927,Y 85.106,Z 90,A 98.302,B 24.9031,C -2.2717,E1 24.9623,E2 -13.3695} C_DIS
LIN {X -15.8025,Y 86.3181,Z 90,A 94.4683,B 24.9031,C -2.2719,E1 24.9728,E2 -9.5316} C_DIS
LIN {X -13.044,Y 86.7782,Z 90,A 92.7735,B 24.9027,C -2.2771,E1 24.9775,E2 -7.8478} C_DIS
LIN {X -10.3193,Y 87.1435,Z 90,A 90.858,B 24.9029,C -2.2745,E1 24.9828,E2 -5.9247} C_DIS
LIN {X -8.1288,Y 87.375,Z 90,A 88.6905,B 24.9048,C -2.2529,E1 24.989,E2 -3.7048} C_DIS
LIN {X -4.158,Y 87.6546,Z 90,A 86.6308,B 24.9033,C -2.2703,E1 24.9946,E2 -1.686} C_DIS
LIN {X -0.7022,Y 87.7496,Z 90,A 84.4856,B 24.903,C -2.2744,E1 25.0006,E2 0.4498} C_DIS
LIN {X 2.6364,Y 87.7127,Z 90,A 82.3224,B 24.9029,C -2.2752,E1 25.0066,E2 2.6108} C_DIS
LIN {X 6.1485,Y 87.5369,Z 90,A 79.9892,B 24.9029,C -2.274,E1 25.0131,E2 4.9457} C_DIS
LIN {X 9.7369,Y 87.2117,Z 90,A 77.7223,B 24.9028,C -2.2764,E1 25.0194,E2 7.2056} C_DIS
LIN {X 12.6022,Y 86.843,Z 90,A 76.0538,B 24.9022,C -2.2829,E1 25.0239,E2 8.8574} C_DIS
LIN {X 15.3756,Y 86.3949,Z 90,A 73.8785,B 24.9032,C -2.2714,E1 25.03,E2 11.0574} C_DIS
LIN {X 19.0475,Y 85.6608,Z 90,A 70.7626,B 24.9051,C -2.2491,E1 25.0387,E2 14.2224} C_DIS
LIN {X 23.1135,Y 84.6539,Z 90,A 69.3639,B 24.9016,C -2.2899,E1 25.0422,E2 15.522} C_DIS
LIN {X 26.3615,Y 83.7,Z 90,A 66.5433,B 24.9034,C -2.2687,E1 25.0498,E2 18.3881} C_DIS
LIN {X 29.1793,Y 82.759,Z 90,A 64.6329,B 24.9035,C -2.2679,E1 25.0549,E2 20.2964} C_DIS
LIN {X 33.8264,Y 80.9711,Z 90,A 61.4101,B 24.9037,C -2.2656,E1 25.0632,E2 23.5176} C_DIS
LIN {X 35.9994,Y 80.0282,Z 90,A 59.9331,B 24.9037,C -2.2662,E1 25.067,E2 24.9896} C_DIS
LIN {X 38.4993,Y 78.8577,Z 90,A 57.7828,B 24.9048,C -2.2526,E1 25.0725,E2 27.1663} C_DIS
LIN {X 42.3274,Y 76.8708,Z 90,A 55.2536,B 24.9043,C -2.2582,E1 25.0786,E2 29.6751} C_DIS
LIN {X 44.9808,Y 75.3481,Z 90,A 52.7415,B 24.906,C -2.2385,E1 25.0848,E2 32.2262} C_DIS
LIN {X 47.9003,Y 73.5269,Z 90,A 50.9575,B 24.905,C -2.2501,E1 25.0889,E2 33.9768} C_DIS
LIN {X 50.3094,Y 71.8992,Z 90,A 48.915,B 24.9057,C -2.2423,E1 25.0936,E2 36.031} C_DIS
LIN {X 54.0113,Y 69.1627,Z 90,A 46.1096,B 24.9056,C -2.2435,E1 25.0998,E2 38.8232} C_DIS
LIN {X 56.3559,Y 67.2651,Z 90,A 43.5072,B 24.9076,C -2.2188,E1 25.1055,E2 41.4739} C_DIS
LIN {X 59.2769,Y 64.7047,Z 90,A 41.3264,B 24.9071,C -2.2256,E1 25.1099,E2 43.6301} C_DIS
LIN {X 61.8148,Y 62.2851,Z 90,A 39.1124,B 24.9073,C -2.2233,E1 25.1143,E2 45.8402} C_DIS
LIN {X 65.5028,Y 58.3941,Z 90,A 35.9063,B 24.9071,C -2.2254,E1 25.1204,E2 49.0271} C_DIS
LIN {X 67.7281,Y 55.7987,Z 90,A 32.9954,B 24.9094,C -2.1974,E1 25.1257,E2 51.9909} C_DIS
LIN {X 70.1368,Y 52.7379,Z 90,A 31.1648,B 24.9079,C -2.2153,E1 25.1287,E2 53.7705} C_DIS
LIN {X 72.3461,Y 49.6665,Z 90,A 28.1885,B 24.9099,C -2.1919,E1 25.1335,E2 56.7875} C_DIS
LIN {X 74.1751,Y 46.8907,Z 90,A 26.5676,B 24.9088,C -2.205,E1 25.1359,E2 58.3694} C_DIS
LIN {X 75.8048,Y 44.2081,Z 90,A 24.3713,B 24.9097,C -2.1945,E1 25.139,E2 60.5792} C_DIS
LIN {X 78.3004,Y 39.6185,Z 90,A 21.1369,B 24.9099,C -2.1913,E1 25.1433,E2 63.8041} C_DIS
LIN {X 79.6934,Y 36.7359,Z 90,A 19.3043,B 24.9097,C -2.1943,E1 25.1454,E2 65.6197} C_DIS
LIN {X 81.2902,Y 33.0509,Z 90,A 16.4704,B 24.9109,C -2.1795,E1 25.1486,E2 68.4731} C_DIS
LIN {X 82.5016,Y 29.8994,Z 90,A 14.406,B 24.911,C -2.1779,E1 25.1506,E2 70.5298} C_DIS
LIN {X 83.9593,Y 25.5252,Z 90,A 11.4325,B 24.9117,C -2.1702,E1 25.1532,E2 73.5046} C_DIS
LIN {X 85.1482,Y 21.2233,Z 90,A 8.3232,B 24.9129,C -2.1545,E1 25.1554,E2 76.633} C_DIS
LIN {X 85.8675,Y 18.0955,Z 90,A 6.1777,B 24.9136,C -2.1463,E1 25.1567,E2 78.7854} C_DIS
LIN {X 86.5561,Y 14.4396,Z 90,A 3.9409,B 24.9136,C -2.1455,E1 25.1578,E2 81.011} C_DIS
LIN {X 87.0264,Y 11.2637,Z 90,A 1.7721,B 24.9144,C -2.1363,E1 25.1586,E2 83.1886} C_DIS
LIN {X 87.3913,Y 7.9515,Z 90,A -0.2848,B 24.9146,C -2.1336,E1 25.1592,E2 85.2398} C_DIS
LIN {X 87.6359,Y 4.5286,Z 90,A -2.6715,B 24.9156,C -2.1214,E1 25.1596,E2 87.6412} C_DIS
LIN {X 87.7476,Y 1.0447,Z 90,A -4.8424,B 24.9159,C -2.1177,E1 25.1598,E2 89.8078} C_DIS
LIN {X 87.7102,Y -2.7167,Z 90,A -7.1681,B 24.9162,C -2.1145,E1 25.1597,E2 92.1273} C_DIS
LIN {X 87.5923,Y -5.3178,Z 90,A -8.9556,B 24.9168,C -2.1059,E1 25.1594,E2 93.9244} C_DIS
LIN {X 87.3774,Y -8.1026,Z 90,A -10.8254,B 24.9174,C -2.0985,E1 25.159,E2 95.8007} C_DIS
LIN {X 86.7504,Y -13.2237,Z 90,A -14.044,B 24.9179,C -2.0929,E1 25.1578,E2 99.0134} C_DIS
LIN {X 86.1106,Y -16.8975,Z 90,A -16.6699,B 24.919,C -2.0785,E1 25.1565,E2 101.658} C_DIS
LIN {X 84.671,Y -23.0502,Z 90,A -21.3883,B 24.9216,C -2.0449,E1 25.1532,E2 106.4284} C_DIS
LIN {X 83.5243,Y -26.9104,Z 90,A -23.3807,B 24.9205,C -2.0588,E1 25.1516,E2 108.3767} C_DIS
LIN {X 82.4063,Y -30.1608,Z 90,A -25.542,B 24.9208,C -2.0547,E1 25.1496,E2 110.5355} C_DIS
LIN {X 80.8104,Y -34.2076,Z 90,A -28.7086,B 24.9224,C -2.0347,E1 25.1462,E2 113.7319} C_DIS
LIN {X 78.1191,Y -39.9733,Z 90,A -32.1871,B 24.9215,C -2.0458,E1 25.142,E2 117.1654} C_DIS
LIN {X 76.1527,Y -43.6032,Z 90,A -35.5565,B 24.9239,C -2.0146,E1 25.1374,E2 120.591} C_DIS
LIN {X 73.9553,Y -47.2347,Z 90,A -38.1797,B 24.9241,C -2.0119,E1 25.1335,E2 123.2073} C_DIS
LIN {X 72.2731,Y -49.7716,Z 90,A -40.7677,B 24.9261,C -1.9858,E1 25.1293,E2 125.8442} C_DIS
LIN {X 69.5664,Y -53.4881,Z 90,A -42.7298,B 24.924,C -2.0133,E1 25.1262,E2 127.7319} C_DIS
LIN {X 66.5969,Y -57.1438,Z 90,A -45.7951,B 24.9246,C -2.0056,E1 25.1207,E2 130.8013} C_DIS
LIN {X 62.2512,Y -61.8491,Z 90,A -49.8667,B 24.9251,C -1.999,E1 25.113,E2 134.8709} C_DIS
LIN {X 59.401,Y -64.5909,Z 90,A -52.6091,B 24.9259,C -1.9873,E1 25.1074,E2 137.6293} C_DIS
LIN {X 54.1938,Y -69.0186,Z 90,A -56.9002,B 24.9263,C -1.9832,E1 25.0982,E2 141.9136} C_DIS
LIN {X 49.7022,Y -72.3213,Z 90,A -60.5139,B 24.9267,C -1.9766,E1 25.09,E2 145.5303} C_DIS
LIN {X 46.8363,Y -74.2091,Z 90,A -63.3247,B 24.9285,C -1.953,E1 25.0833,E2 148.3876} C_DIS
LIN {X 42.4093,Y -76.8247,Z 90,A -66.6565,B 24.9289,C -1.9479,E1 25.0752,E2 151.7217} C_DIS
LIN {X 35.9122,Y -80.0675,Z 90,A -70.9496,B 24.9283,C -1.9553,E1 25.0645,E2 155.986} C_DIS
LIN {X 32.6159,Y -81.4673,Z 90,A -73.2931,B 24.9286,C -1.9517,E1 25.0584,E2 158.3324} C_DIS
LIN {X 28.8365,Y -82.8793,Z 90,A -76.0882,B 24.9292,C -1.943,E1 25.0511,E2 161.1425} C_DIS
LIN {X 23.2729,Y -84.6108,Z 90,A -79.757,B 24.9292,C -1.943,E1 25.0413,E2 164.8046} C_DIS
LIN {X 20.8876,Y -85.2301,Z 90,A -82.3288,B 24.9316,C -1.9102,E1 25.0341,E2 167.4505} C_DIS
LIN {X 16.1293,Y -86.2585,Z 90,A -84.521,B 24.9295,C -1.9394,E1 25.0283,E2 169.5709} C_DIS
LIN {X 13.0796,Y -86.7727,Z 90,A -86.4789,B 24.9295,C -1.94,E1 25.0229,E2 171.5256} C_DIS
LIN {X 8.9431,Y -87.2956,Z 90,A -89.1368,B 24.9295,C -1.9404,E1 25.0155,E2 174.1805} C_DIS
LIN {X 6.3088,Y -87.5261,Z 90,A -90.9431,B 24.9297,C -1.937,E1 25.0105,E2 175.9941} C_DIS
LIN {X 3.6059,Y -87.6783,Z 90,A -92.7651,B 24.9298,C -1.9345,E1 25.0054,E2 177.8211} C_DIS
LIN {X 0.5814,Y -87.7407,Z 90,A -94.2372,B 24.9287,C -1.9503,E1 25.0014,E2 179.2555} C_DIS
Enddeposition()
LIN {X 0.5814,Y -87.7407,Z 90,A -94.2372,B 24.9287,C -1.9503,E1 25.0014,E2 179.2555} C_DIS
Startdeposition()
$VEL.CP = VEL_PRINT
LIN {X 2.486,Y -86.7363,Z 90,A -92.5164,B 24.9263,C -1.9825,E1 25.0064,E2 177.4588} C_DIS
LIN {X 5.0865,Y -86.623,Z 90,A -90.7531,B 24.9262,C -1.9846,E1 25.0113,E2 175.6911} C_DIS
LIN {X 8.5234,Y -86.3536,Z 90,A -88.6941,B 24.9266,C -1.9787,E1 25.017,E2 173.6473} C_DIS
LIN {X 11.6055,Y -85.9934,Z 90,A -86.6801,B 24.9266,C -1.9788,E1 25.0226,E2 171.6345} C_DIS
Enddeposition()
END
